LIN {X 0,Y 549.167,Z 589.017,A -85,B 0,C 180,E1 -11279.852,E2 -11279.852} C_VEL
LIN {X 0,Y 549.143,Z 589.013,A -85,B 0,C 180,E1 -11282.665,E2 -11282.665} C_VEL
LIN {X 0,Y 549.213,Z 589.004,A -85,B 0,C 180,E1 -11285.921,E2 -11285.921} C_VEL
LIN {X 0,Y 549.155,Z 589.006,A -85,B 0,C 180,E1 -11288.918,E2 -11288.918} C_VEL
LIN {X 0,Y 549.152,Z 589.01,A -85,B 0,C 180,E1 -11291.549,E2 -11291.549} C_VEL
LIN {X 0,Y 549.201,Z 589.004,A -85,B 0,C 180,E1 -11294.545,E2 -11294.545} C_VEL
LIN {X 0,Y 549.18,Z 589.01,A -85,B 0,C 180,E1 -11297.711,E2 -11297.711} C_VEL
LIN {X 0,Y 549.182,Z 589.007,A -85,B 0,C 180,E1 -11300.378,E2 -11300.378} C_VEL
LIN {X 0,Y 549.209,Z 589.006,A -85,B 0,C 180,E1 -11303.464,E2 -11303.464} C_VEL
LIN {X 0,Y 549.192,Z 589.005,A -85,B 0,C 180,E1 -11305.998,E2 -11305.998} C_VEL
LIN {X 0,Y 549.178,Z 589.011,A -85,B 0,C 180,E1 -11308.71,E2 -11308.71} C_VEL
LIN {X 0,Y 549.192,Z 589.009,A -85,B 0,C 180,E1 -11311.01,E2 -11311.01} C_VEL
LIN {X 0,Y 549.177,Z 589.009,A -85,B 0,C 180,E1 -11313.487,E2 -11313.487} C_VEL
LIN {X 0,Y 549.182,Z 589.008,A -85,B 0,C 180,E1 -11315.912,E2 -11315.912} C_VEL
LIN {X 0,Y 549.213,Z 589.011,A -85,B 0,C 180,E1 -11318.594,E2 -11318.594} C_VEL
LIN {X 0,Y 549.193,Z 589.011,A -85,B 0,C 180,E1 -11321.406,E2 -11321.406} C_VEL
LIN {X 0,Y 549.206,Z 589.008,A -85,B 0,C 180,E1 -11323.705,E2 -11323.705} C_VEL
LIN {X 0,Y 549.285,Z 588.998,A -85,B 0,C 180,E1 -11325.978,E2 -11325.978} C_VEL
LIN {X 0,Y 549.266,Z 589.108,A -85,B 0,C 180,E1 -11328.087,E2 -11328.087} C_VEL
LIN {X 0,Y 551,Z 598.292,A -85,B 0,C 180,E1 -11330.118,E2 -11330.118} C_VEL
LIN {X 0,Y 551.12,Z 603.64,A -85,B 0,C 180,E1 -11331.227,E2 -11331.227} C_VEL
LIN {X 0,Y 550.41,Z 616.517,A -85,B 0,C 180,E1 -11333.79,E2 -11333.79} C_VEL
LIN {X 0,Y 549.829,Z 624.477,A -85,B 0,C 180,E1 -11335.341,E2 -11335.341} C_VEL
LIN {X 0,Y 553.064,Z 642.479,A -85,B 0,C 180,E1 -11335.755,E2 -11335.755} C_VEL
LIN {X 0,Y 551.552,Z 730.311,A -85,B 0,C 180,E1 -11337.111,E2 -11337.111} C_VEL
LIN {X 0,Y 551.333,Z 739.943,A -85,B 0,C 180,E1 -11337.337,E2 -11337.337} C_VEL
LIN {X 0,Y 551.078,Z 750.352,A -85,B 0,C 180,E1 -11337.678,E2 -11337.678} C_VEL
LIN {X 0,Y 550.845,Z 759.981,A -85,B 0,C 180,E1 -11338.087,E2 -11338.087} C_VEL
LIN {X 0,Y 550.538,Z 770.195,A -85,B 0,C 180,E1 -11338.633,E2 -11338.633} C_VEL
LIN {X 0,Y 550.186,Z 779.879,A -85,B 0,C 180,E1 -11339.27,E2 -11339.27} C_VEL
LIN {X 0,Y 549.809,Z 788.022,A -85,B 0,C 180,E1 -11339.909,E2 -11339.909} C_VEL
LIN {X 0,Y 549.317,Z 796.766,A -85,B 0,C 180,E1 -11340.73,E2 -11340.73} C_VEL
LIN {X 0,Y 548.892,Z 803.411,A -85,B 0,C 180,E1 -11341.462,E2 -11341.462} C_VEL
LIN {X 0,Y 548.614,Z 810.348,A -85,B 0,C 180,E1 -11342.378,E2 -11342.378} C_VEL
LIN {X 0,Y 548.231,Z 816.184,A -85,B 0,C 180,E1 -11343.296,E2 -11343.296} C_VEL
LIN {X 0,Y 548.099,Z 822.583,A -85,B 0,C 180,E1 -11344.579,E2 -11344.579} C_VEL
LIN {X 0,Y 547.955,Z 827.199,A -85,B 0,C 180,E1 -11345.793,E2 -11345.793} C_VEL
LIN {X 0,Y 547.864,Z 829.635,A -85,B 0,C 180,E1 -11346.607,E2 -11346.607} C_VEL
LIN {X 0,Y 547.753,Z 831.287,A -85,B 0,C 180,E1 -11347.347,E2 -11347.347} C_VEL
LIN {X 0,Y 547.692,Z 833.366,A -85,B 0,C 180,E1 -11348.828,E2 -11348.828} C_VEL
LIN {X 0,Y 547.683,Z 833.621,A -85,B 0,C 180,E1 -11350.314,E2 -11350.314} C_VEL
LIN {X 0,Y 547.698,Z 833.236,A -85,B 0,C 180,E1 -11351.059,E2 -11351.059} C_VEL
LIN {X 0,Y 547.699,Z 830.896,A -85,B 0,C 180,E1 -11352.557,E2 -11352.557} C_VEL
LIN {X 0,Y 547.84,Z 828.07,A -85,B 0,C 180,E1 -11353.662,E2 -11353.662} C_VEL
LIN {X 0,Y 547.893,Z 825.548,A -85,B 0,C 180,E1 -11354.435,E2 -11354.435} C_VEL
LIN {X 0,Y 548.091,Z 819.726,A -85,B 0,C 180,E1 -11355.757,E2 -11355.757} C_VEL
LIN {X 0,Y 548.25,Z 814.051,A -85,B 0,C 180,E1 -11356.773,E2 -11356.773} C_VEL
LIN {X 0,Y 548.469,Z 808.116,A -85,B 0,C 180,E1 -11357.656,E2 -11357.656} C_VEL
LIN {X 0,Y 548.826,Z 800.373,A -85,B 0,C 180,E1 -11358.606,E2 -11358.606} C_VEL
LIN {X 0,Y 549.141,Z 791.937,A -85,B 0,C 180,E1 -11359.465,E2 -11359.465} C_VEL
LIN {X 0,Y 549.465,Z 782.896,A -85,B 0,C 180,E1 -11360.229,E2 -11360.229} C_VEL
LIN {X 0,Y 549.851,Z 773.343,A -85,B 0,C 180,E1 -11360.896,E2 -11360.896} C_VEL
LIN {X 0,Y 550.162,Z 765.257,A -85,B 0,C 180,E1 -11361.373,E2 -11361.373} C_VEL
LIN {X 0,Y 550.473,Z 753.781,A -85,B 0,C 180,E1 -11361.91,E2 -11361.91} C_VEL
LIN {X 0,Y 550.673,Z 742.561,A -85,B 0,C 180,E1 -11362.31,E2 -11362.31} C_VEL
LIN {X 0,Y 550.9,Z 732.608,A -85,B 0,C 180,E1 -11362.57,E2 -11362.57} C_VEL
LIN {X 0,Y 551.202,Z 713.558,A -85,B 0,C 180,E1 -11362.878,E2 -11362.878} C_VEL
LIN {X 0,Y 551.969,Z 640.723,A -85,B 0,C 180,E1 -11363.953,E2 -11363.953} C_VEL
LIN {X 0,Y 549.342,Z 623.321,A -85,B 0,C 180,E1 -11364.283,E2 -11364.283} C_VEL
LIN {X 0,Y 550.029,Z 607.305,A -85,B 0,C 180,E1 -11367.287,E2 -11367.287} C_VEL
LIN {X 0,Y 550.372,Z 596.511,A -85,B 0,C 180,E1 -11369.339,E2 -11369.339} C_VEL
LIN {X 0,Y 549.276,Z 588.999,A -85,B 0,C 180,E1 -11370.871,E2 -11370.871} C_VEL
LIN {X 0,Y 549.193,Z 589.009,A -85,B 0,C 180,E1 -11374.137,E2 -11374.137} C_VEL
LIN {X 0,Y 549.19,Z 589.003,A -85,B 0,C 180,E1 -11376.83,E2 -11376.83} C_VEL
LIN {X 0,Y 549.2,Z 589.009,A -85,B 0,C 180,E1 -11380.072,E2 -11380.072} C_VEL
LIN {X 0,Y 549.187,Z 589.005,A -85,B 0,C 180,E1 -11383.365,E2 -11383.365} C_VEL
LIN {X 0,Y 549.195,Z 589.006,A -85,B 0,C 180,E1 -11385.579,E2 -11385.579} C_VEL
LIN {X 0,Y 549.173,Z 589.005,A -85,B 0,C 180,E1 -11388.808,E2 -11388.808} C_VEL
LIN {X 0,Y 549.149,Z 589.009,A -85,B 0,C 180,E1 -11391.318,E2 -11391.318} C_VEL
LIN {X 0,Y 549.236,Z 589.005,A -85,B 0,C 180,E1 -11394.081,E2 -11394.081} C_VEL
LIN {X 0,Y 549.162,Z 589.007,A -85,B 0,C 180,E1 -11396.739,E2 -11396.739} C_VEL
LIN {X 0,Y 549.177,Z 589.005,A -85,B 0,C 180,E1 -11399.324,E2 -11399.324} C_VEL
LIN {X 0,Y 549.202,Z 589.009,A -85,B 0,C 180,E1 -11401.843,E2 -11401.843} C_VEL
LIN {X 0,Y 549.169,Z 589.005,A -85,B 0,C 180,E1 -11404.9,E2 -11404.9} C_VEL
LIN {X 0,Y 549.197,Z 589.005,A -85,B 0,C 180,E1 -11407.504,E2 -11407.504} C_VEL
LIN {X 0,Y 549.19,Z 589.01,A -85,B 0,C 180,E1 -11409.857,E2 -11409.857} C_VEL
LIN {X 0,Y 549.225,Z 588.998,A -85,B 0,C 180,E1 -11413.036,E2 -11413.036} C_VEL
LIN {X 0,Y 549.283,Z 589.001,A -85,B 0,C 180,E1 -11415.978,E2 -11415.978} C_VEL
LIN {X 0,Y 549.241,Z 588.998,A -85,B 0,C 180,E1 -11416.542,E2 -11416.542} C_VEL
LIN {X 0,Y 548.584,Z 589.079,A -85,B 0,C 180,E1 -11417.154,E2 -11417.154} C_VEL
LIN {X 0,Y 545.779,Z 589.434,A -85,B 0,C 180,E1 -11418.148,E2 -11418.148} C_VEL
LIN {X 0,Y 543.388,Z 589.731,A -85,B 0,C 180,E1 -11418.948,E2 -11418.948} C_VEL
LIN {X 0,Y 542.33,Z 589.861,A -85,B 0,C 180,E1 -11419.565,E2 -11419.565} C_VEL
LIN {X 0,Y 542.226,Z 589.873,A -85,B 0,C 180,E1 -11419.774,E2 -11419.774} C_VEL
LIN {X 0,Y 542.282,Z 589.865,A -85,B 0,C 180,E1 -11422.578,E2 -11422.578} C_VEL
LIN {X 0,Y 542.347,Z 589.855,A -85,B 0,C 180,E1 -11424.813,E2 -11424.813} C_VEL
LIN {X 0,Y 542.15,Z 589.88,A -85,B 0,C 180,E1 -11427.038,E2 -11427.038} C_VEL
LIN {X 0,Y 542.498,Z 589.846,A -85,B 0,C 180,E1 -11430,E2 -11430} C_VEL
LIN {X 0,Y 542.313,Z 589.865,A -85,B 0,C 180,E1 -11433.703,E2 -11433.703} C_VEL
LIN {X 0,Y 542.34,Z 589.865,A -85,B 0,C 180,E1 -11436.033,E2 -11436.033} C_VEL
LIN {X 0,Y 542.226,Z 589.87,A -85,B 0,C 180,E1 -11438.918,E2 -11438.918} C_VEL
LIN {X 0,Y 542.235,Z 589.869,A -85,B 0,C 180,E1 -11441.173,E2 -11441.173} C_VEL
LIN {X 0,Y 542.236,Z 589.873,A -85,B 0,C 180,E1 -11444.346,E2 -11444.346} C_VEL
LIN {X 0,Y 542.17,Z 589.878,A -85,B 0,C 180,E1 -11447.286,E2 -11447.286} C_VEL
LIN {X 0,Y 542.161,Z 589.881,A -85,B 0,C 180,E1 -11450.415,E2 -11450.415} C_VEL
LIN {X 0,Y 542.138,Z 589.881,A -85,B 0,C 180,E1 -11452.805,E2 -11452.805} C_VEL
LIN {X 0,Y 542.134,Z 589.882,A -85,B 0,C 180,E1 -11455.258,E2 -11455.258} C_VEL
LIN {X 0,Y 542.151,Z 589.885,A -85,B 0,C 180,E1 -11457.717,E2 -11457.717} C_VEL
LIN {X 0,Y 542.149,Z 589.885,A -85,B 0,C 180,E1 -11460.256,E2 -11460.256} C_VEL
LIN {X 0,Y 542.129,Z 589.882,A -85,B 0,C 180,E1 -11462.88,E2 -11462.88} C_VEL
LIN {X 0,Y 542.188,Z 589.878,A -85,B 0,C 180,E1 -11465.545,E2 -11465.545} C_VEL
LIN {X 0,Y 542.123,Z 589.887,A -85,B 0,C 180,E1 -11468.329,E2 -11468.329} C_VEL
LIN {X 0,Y 542.125,Z 589.883,A -85,B 0,C 180,E1 -11471.219,E2 -11471.219} C_VEL
LIN {X 0,Y 542.15,Z 589.885,A -85,B 0,C 180,E1 -11474.24,E2 -11474.24} C_VEL
LIN {X 0,Y 542.127,Z 589.883,A -85,B 0,C 180,E1 -11476.783,E2 -11476.783} C_VEL
LIN {X 0,Y 542.153,Z 589.885,A -85,B 0,C 180,E1 -11479.761,E2 -11479.761} C_VEL
LIN {X 0,Y 542.165,Z 589.879,A -85,B 0,C 180,E1 -11482.612,E2 -11482.612} C_VEL
LIN {X 0,Y 542.155,Z 589.881,A -85,B 0,C 180,E1 -11485.357,E2 -11485.357} C_VEL
LIN {X 0,Y 542.125,Z 589.885,A -85,B 0,C 180,E1 -11488.511,E2 -11488.511} C_VEL
LIN {X 0,Y 542.142,Z 589.883,A -85,B 0,C 180,E1 -11491.468,E2 -11491.468} C_VEL
LIN {X 0,Y 542.111,Z 589.894,A -85,B 0,C 180,E1 -11493.941,E2 -11493.941} C_VEL
LIN {X 0,Y 542.138,Z 589.883,A -85,B 0,C 180,E1 -11496.538,E2 -11496.538} C_VEL
LIN {X 0,Y 542.165,Z 589.878,A -85,B 0,C 180,E1 -11498.793,E2 -11498.793} C_VEL
LIN {X 0,Y 542.15,Z 589.88,A -85,B 0,C 180,E1 -11501.156,E2 -11501.156} C_VEL
LIN {X 0,Y 542.164,Z 589.881,A -85,B 0,C 180,E1 -11503.488,E2 -11503.488} C_VEL
LIN {X 0,Y 542.242,Z 589.875,A -85,B 0,C 180,E1 -11505.793,E2 -11505.793} C_VEL
LIN {X 0,Y 542.279,Z 589.864,A -85,B 0,C 180,E1 -11509.012,E2 -11509.012} C_VEL
LIN {X 0,Y 542.263,Z 589.873,A -85,B 0,C 180,E1 -11511.832,E2 -11511.832} C_VEL
LIN {X 0,Y 542.352,Z 589.862,A -85,B 0,C 180,E1 -11514.07,E2 -11514.07} C_VEL
LIN {X 0,Y 542.308,Z 589.864,A -85,B 0,C 180,E1 -11516.298,E2 -11516.298} C_VEL
LIN {X 0,Y 542.502,Z 589.845,A -85,B 0,C 180,E1 -11520,E2 -11520} C_VEL
LIN {X 0,Y 542.306,Z 589.866,A -85,B 0,C 180,E1 -11523.703,E2 -11523.703} C_VEL
LIN {X 0,Y 542.364,Z 589.861,A -85,B 0,C 180,E1 -11526.052,E2 -11526.052} C_VEL
LIN {X 0,Y 542.233,Z 589.869,A -85,B 0,C 180,E1 -11528.918,E2 -11528.918} C_VEL
LIN {X 0,Y 542.238,Z 589.869,A -85,B 0,C 180,E1 -11531.173,E2 -11531.173} C_VEL
LIN {X 0,Y 542.227,Z 589.874,A -85,B 0,C 180,E1 -11534.34,E2 -11534.34} C_VEL
LIN {X 0,Y 542.136,Z 589.883,A -85,B 0,C 180,E1 -11537.287,E2 -11537.287} C_VEL
LIN {X 0,Y 542.139,Z 589.885,A -85,B 0,C 180,E1 -11539.629,E2 -11539.629} C_VEL
LIN {X 0,Y 542.124,Z 589.892,A -85,B 0,C 180,E1 -11542.005,E2 -11542.005} C_VEL
LIN {X 0,Y 542.137,Z 589.884,A -85,B 0,C 180,E1 -11544.421,E2 -11544.421} C_VEL
LIN {X 0,Y 542.154,Z 589.885,A -85,B 0,C 180,E1 -11547.717,E2 -11547.717} C_VEL
LIN {X 0,Y 542.121,Z 589.888,A -85,B 0,C 180,E1 -11550.258,E2 -11550.258} C_VEL
LIN {X 0,Y 542.112,Z 589.885,A -85,B 0,C 180,E1 -11552.877,E2 -11552.877} C_VEL
LIN {X 0,Y 542.121,Z 589.887,A -85,B 0,C 180,E1 -11555.55,E2 -11555.55} C_VEL
LIN {X 0,Y 542.088,Z 589.891,A -85,B 0,C 180,E1 -11558.332,E2 -11558.332} C_VEL
LIN {X 0,Y 542.13,Z 589.885,A -85,B 0,C 180,E1 -11561.464,E2 -11561.464} C_VEL
LIN {X 0,Y 542.149,Z 589.88,A -85,B 0,C 180,E1 -11564.717,E2 -11564.717} C_VEL
LIN {X 0,Y 542.103,Z 589.888,A -85,B 0,C 180,E1 -11567.433,E2 -11567.433} C_VEL
LIN {X 0,Y 542.116,Z 589.89,A -85,B 0,C 180,E1 -11569.757,E2 -11569.757} C_VEL
LIN {X 0,Y 542.1,Z 589.887,A -85,B 0,C 180,E1 -11572.607,E2 -11572.607} C_VEL
LIN {X 0,Y 542.12,Z 589.885,A -85,B 0,C 180,E1 -11575.354,E2 -11575.354} C_VEL
LIN {X 0,Y 542.109,Z 589.894,A -85,B 0,C 180,E1 -11578.012,E2 -11578.012} C_VEL
LIN {X 0,Y 542.139,Z 589.882,A -85,B 0,C 180,E1 -11580.596,E2 -11580.596} C_VEL
LIN {X 0,Y 542.116,Z 589.884,A -85,B 0,C 180,E1 -11583.114,E2 -11583.114} C_VEL
LIN {X 0,Y 542.153,Z 589.943,A -85,B 0,C 180,E1 -11585.935,E2 -11585.935} C_VEL
LIN {X 0,Y 544.262,Z 601.967,A -85,B 0,C 180,E1 -11588.086,E2 -11588.086} C_VEL
LIN {X 0,Y 543.789,Z 613.914,A -85,B 0,C 180,E1 -11590.102,E2 -11590.102} C_VEL
LIN {X 0,Y 542.762,Z 634.369,A -85,B 0,C 180,E1 -11593.506,E2 -11593.506} C_VEL
LIN {X 0,Y 542.247,Z 647.24,A -85,B 0,C 180,E1 -11595.592,E2 -11595.592} C_VEL
LIN {X 0,Y 544.925,Z 670.18,A -85,B 0,C 180,E1 -11596.006,E2 -11596.006} C_VEL
LIN {X 0,Y 543.974,Z 754.194,A -85,B 0,C 180,E1 -11597.285,E2 -11597.285} C_VEL
LIN {X 0,Y 543.75,Z 763.983,A -85,B 0,C 180,E1 -11597.516,E2 -11597.516} C_VEL
LIN {X 0,Y 543.475,Z 773.356,A -85,B 0,C 180,E1 -11597.817,E2 -11597.817} C_VEL
LIN {X 0,Y 543.155,Z 784.221,A -85,B 0,C 180,E1 -11598.277,E2 -11598.277} C_VEL
LIN {X 0,Y 542.941,Z 792.736,A -85,B 0,C 180,E1 -11598.722,E2 -11598.722} C_VEL
LIN {X 0,Y 542.524,Z 803.182,A -85,B 0,C 180,E1 -11599.398,E2 -11599.398} C_VEL
LIN {X 0,Y 542.148,Z 812.599,A -85,B 0,C 180,E1 -11600.143,E2 -11600.143} C_VEL
LIN {X 0,Y 541.76,Z 820.502,A -85,B 0,C 180,E1 -11600.887,E2 -11600.887} C_VEL
LIN {X 0,Y 541.379,Z 828.715,A -85,B 0,C 180,E1 -11601.818,E2 -11601.818} C_VEL
LIN {X 0,Y 541.142,Z 835.553,A -85,B 0,C 180,E1 -11602.75,E2 -11602.75} C_VEL
LIN {X 0,Y 540.958,Z 841.257,A -85,B 0,C 180,E1 -11603.681,E2 -11603.681} C_VEL
LIN {X 0,Y 540.832,Z 846.778,A -85,B 0,C 180,E1 -11604.799,E2 -11604.799} C_VEL
LIN {X 0,Y 540.736,Z 849.867,A -85,B 0,C 180,E1 -11605.543,E2 -11605.543} C_VEL
LIN {X 0,Y 540.68,Z 853.432,A -85,B 0,C 180,E1 -11606.658,E2 -11606.658} C_VEL
LIN {X 0,Y 540.682,Z 855.954,A -85,B 0,C 180,E1 -11607.773,E2 -11607.773} C_VEL
LIN {X 0,Y 540.646,Z 857.752,A -85,B 0,C 180,E1 -11609.258,E2 -11609.258} C_VEL
LIN {X 0,Y 540.635,Z 858.065,A -85,B 0,C 180,E1 -11610,E2 -11610} C_VEL
LIN {X 0,Y 540.647,Z 857.414,A -85,B 0,C 180,E1 -11611.485,E2 -11611.485} C_VEL
LIN {X 0,Y 540.682,Z 856.4,A -85,B 0,C 180,E1 -11612.227,E2 -11612.227} C_VEL
LIN {X 0,Y 540.712,Z 853.243,A -85,B 0,C 180,E1 -11613.714,E2 -11613.714} C_VEL
LIN {X 0,Y 540.783,Z 849.623,A -85,B 0,C 180,E1 -11614.83,E2 -11614.83} C_VEL
LIN {X 0,Y 540.937,Z 844.88,A -85,B 0,C 180,E1 -11615.946,E2 -11615.946} C_VEL
LIN {X 0,Y 541.151,Z 838.85,A -85,B 0,C 180,E1 -11617.063,E2 -11617.063} C_VEL
LIN {X 0,Y 541.488,Z 831.311,A -85,B 0,C 180,E1 -11618.181,E2 -11618.181} C_VEL
LIN {X 0,Y 541.88,Z 823.679,A -85,B 0,C 180,E1 -11619.111,E2 -11619.111} C_VEL
LIN {X 0,Y 542.348,Z 815.452,A -85,B 0,C 180,E1 -11619.947,E2 -11619.947} C_VEL
LIN {X 0,Y 542.781,Z 806.721,A -85,B 0,C 180,E1 -11620.691,E2 -11620.691} C_VEL
LIN {X 0,Y 543.202,Z 797.041,A -85,B 0,C 180,E1 -11621.375,E2 -11621.375} C_VEL
LIN {X 0,Y 543.603,Z 788.118,A -85,B 0,C 180,E1 -11621.898,E2 -11621.898} C_VEL
LIN {X 0,Y 544.02,Z 777.27,A -85,B 0,C 180,E1 -11622.407,E2 -11622.407} C_VEL
LIN {X 0,Y 544.358,Z 767.174,A -85,B 0,C 180,E1 -11622.777,E2 -11622.777} C_VEL
LIN {X 0,Y 544.713,Z 755.878,A -85,B 0,C 180,E1 -11623.076,E2 -11623.076} C_VEL
LIN {X 0,Y 545.07,Z 733.637,A -85,B 0,C 180,E1 -11623.445,E2 -11623.445} C_VEL
LIN {X 0,Y 545.976,Z 669.088,A -85,B 0,C 180,E1 -11624.461,E2 -11624.461} C_VEL
LIN {X 0,Y 543.573,Z 651.51,A -85,B 0,C 180,E1 -11624.84,E2 -11624.84} C_VEL
LIN {X 0,Y 542.613,Z 645.876,A -85,B 0,C 180,E1 -11624.986,E2 -11624.986} C_VEL
LIN {X 0,Y 543.607,Z 626.95,A -85,B 0,C 180,E1 -11628.208,E2 -11628.208} C_VEL
LIN {X 0,Y 544.885,Z 608.18,A -85,B 0,C 180,E1 -11631.492,E2 -11631.492} C_VEL
LIN {X 0,Y 544.87,Z 604.061,A -85,B 0,C 180,E1 -11632.244,E2 -11632.244} C_VEL
LIN {X 0,Y 542.428,Z 591.113,A -85,B 0,C 180,E1 -11634.814,E2 -11634.814} C_VEL
LIN {X 0,Y 542.136,Z 589.89,A -85,B 0,C 180,E1 -11635.104,E2 -11635.104} C_VEL
LIN {X 0,Y 542.131,Z 589.895,A -85,B 0,C 180,E1 -11637.719,E2 -11637.719} C_VEL
LIN {X 0,Y 542.121,Z 589.89,A -85,B 0,C 180,E1 -11640.258,E2 -11640.258} C_VEL
LIN {X 0,Y 542.113,Z 589.89,A -85,B 0,C 180,E1 -11642.877,E2 -11642.877} C_VEL
LIN {X 0,Y 542.164,Z 589.885,A -85,B 0,C 180,E1 -11645.547,E2 -11645.547} C_VEL
LIN {X 0,Y 542.102,Z 589.883,A -85,B 0,C 180,E1 -11648.331,E2 -11648.331} C_VEL
LIN {X 0,Y 542.133,Z 589.884,A -85,B 0,C 180,E1 -11651.464,E2 -11651.464} C_VEL
LIN {X 0,Y 542.154,Z 589.881,A -85,B 0,C 180,E1 -11654.24,E2 -11654.24} C_VEL
LIN {X 0,Y 542.156,Z 589.885,A -85,B 0,C 180,E1 -11656.785,E2 -11656.785} C_VEL
LIN {X 0,Y 542.157,Z 589.883,A -85,B 0,C 180,E1 -11659.761,E2 -11659.761} C_VEL
LIN {X 0,Y 542.168,Z 589.886,A -85,B 0,C 180,E1 -11663.226,E2 -11663.226} C_VEL
LIN {X 0,Y 542.147,Z 589.883,A -85,B 0,C 180,E1 -11665.779,E2 -11665.779} C_VEL
LIN {X 0,Y 542.128,Z 589.892,A -85,B 0,C 180,E1 -11668.881,E2 -11668.881} C_VEL
LIN {X 0,Y 542.146,Z 589.884,A -85,B 0,C 180,E1 -11671.468,E2 -11671.468} C_VEL
LIN {X 0,Y 542.112,Z 589.889,A -85,B 0,C 180,E1 -11673.941,E2 -11673.941} C_VEL
LIN {X 0,Y 542.143,Z 589.891,A -85,B 0,C 180,E1 -11676.537,E2 -11676.537} C_VEL
LIN {X 0,Y 542.164,Z 589.885,A -85,B 0,C 180,E1 -11679.584,E2 -11679.584} C_VEL
LIN {X 0,Y 542.155,Z 589.889,A -85,B 0,C 180,E1 -11681.936,E2 -11681.936} C_VEL
LIN {X 0,Y 542.206,Z 589.88,A -85,B 0,C 180,E1 -11685.027,E2 -11685.027} C_VEL
LIN {X 0,Y 542.244,Z 589.98,A -85,B 0,C 180,E1 -11687.835,E2 -11687.835} C_VEL
LIN {X 0,Y 544.06,Z 599.517,A -85,B 0,C 180,E1 -11689.991,E2 -11689.991} C_VEL
LIN {X 0,Y 544.203,Z 604.855,A -85,B 0,C 180,E1 -11691.115,E2 -11691.115} C_VEL
LIN {X 0,Y 543.453,Z 617.675,A -85,B 0,C 180,E1 -11693.71,E2 -11693.71} C_VEL
LIN {X 0,Y 542.906,Z 624.687,A -85,B 0,C 180,E1 -11695.097,E2 -11695.097} C_VEL
LIN {X 0,Y 546.289,Z 642.987,A -85,B 0,C 180,E1 -11695.53,E2 -11695.53} C_VEL
LIN {X 0,Y 545.008,Z 710.544,A -85,B 0,C 180,E1 -11696.592,E2 -11696.592} C_VEL
LIN {X 0,Y 544.667,Z 732.534,A -85,B 0,C 180,E1 -11696.959,E2 -11696.959} C_VEL
LIN {X 0,Y 544.359,Z 745.377,A -85,B 0,C 180,E1 -11697.303,E2 -11697.303} C_VEL
LIN {X 0,Y 543.974,Z 759.583,A -85,B 0,C 180,E1 -11697.878,E2 -11697.878} C_VEL
LIN {X 0,Y 543.646,Z 769.909,A -85,B 0,C 180,E1 -11698.431,E2 -11698.431} C_VEL
LIN {X 0,Y 543.309,Z 779.666,A -85,B 0,C 180,E1 -11699.076,E2 -11699.076} C_VEL
LIN {X 0,Y 542.822,Z 788.904,A -85,B 0,C 180,E1 -11699.815,E2 -11699.815} C_VEL
LIN {X 0,Y 542.376,Z 796.687,A -85,B 0,C 180,E1 -11700.555,E2 -11700.555} C_VEL
LIN {X 0,Y 541.835,Z 804.804,A -85,B 0,C 180,E1 -11701.481,E2 -11701.481} C_VEL
LIN {X 0,Y 541.545,Z 811.542,A -85,B 0,C 180,E1 -11702.409,E2 -11702.409} C_VEL
LIN {X 0,Y 541.159,Z 817.201,A -85,B 0,C 180,E1 -11703.339,E2 -11703.339} C_VEL
LIN {X 0,Y 541.067,Z 822.652,A -85,B 0,C 180,E1 -11704.455,E2 -11704.455} C_VEL
LIN {X 0,Y 540.901,Z 826.94,A -85,B 0,C 180,E1 -11705.573,E2 -11705.573} C_VEL
LIN {X 0,Y 540.76,Z 830.153,A -85,B 0,C 180,E1 -11706.694,E2 -11706.694} C_VEL
LIN {X 0,Y 540.644,Z 831.8,A -85,B 0,C 180,E1 -11707.444,E2 -11707.444} C_VEL
LIN {X 0,Y 540.593,Z 833.6,A -85,B 0,C 180,E1 -11708.945,E2 -11708.945} C_VEL
LIN {X 0,Y 540.618,Z 833.9,A -85,B 0,C 180,E1 -11710.039,E2 -11710.039} C_VEL
LIN {X 0,Y 540.601,Z 833.202,A -85,B 0,C 180,E1 -11711.207,E2 -11711.207} C_VEL
LIN {X 0,Y 540.556,Z 832.172,A -85,B 0,C 180,E1 -11711.965,E2 -11711.965} C_VEL
LIN {X 0,Y 540.733,Z 828.837,A -85,B 0,C 180,E1 -11713.483,E2 -11713.483} C_VEL
LIN {X 0,Y 540.825,Z 825.024,A -85,B 0,C 180,E1 -11714.628,E2 -11714.628} C_VEL
LIN {X 0,Y 541.005,Z 819.977,A -85,B 0,C 180,E1 -11715.776,E2 -11715.776} C_VEL
LIN {X 0,Y 541.159,Z 814.982,A -85,B 0,C 180,E1 -11716.701,E2 -11716.701} C_VEL
LIN {X 0,Y 541.399,Z 808.392,A -85,B 0,C 180,E1 -11717.7,E2 -11717.7} C_VEL
LIN {X 0,Y 541.758,Z 800.663,A -85,B 0,C 180,E1 -11718.662,E2 -11718.662} C_VEL
LIN {X 0,Y 542.075,Z 793.055,A -85,B 0,C 180,E1 -11719.459,E2 -11719.459} C_VEL
LIN {X 0,Y 542.412,Z 783.227,A -85,B 0,C 180,E1 -11720.307,E2 -11720.307} C_VEL
LIN {X 0,Y 542.831,Z 773.716,A -85,B 0,C 180,E1 -11720.982,E2 -11720.982} C_VEL
LIN {X 0,Y 543.155,Z 764.302,A -85,B 0,C 180,E1 -11721.534,E2 -11721.534} C_VEL
LIN {X 0,Y 543.475,Z 754.567,A -85,B 0,C 180,E1 -11721.997,E2 -11721.997} C_VEL
LIN {X 0,Y 543.669,Z 743.239,A -85,B 0,C 180,E1 -11722.412,E2 -11722.412} C_VEL
LIN {X 0,Y 543.91,Z 732.23,A -85,B 0,C 180,E1 -11722.701,E2 -11722.701} C_VEL
LIN {X 0,Y 544.239,Z 713.189,A -85,B 0,C 180,E1 -11723.012,E2 -11723.012} C_VEL
LIN {X 0,Y 545.027,Z 641.328,A -85,B 0,C 180,E1 -11724.09,E2 -11724.09} C_VEL
LIN {X 0,Y 542.333,Z 623.472,A -85,B 0,C 180,E1 -11724.437,E2 -11724.437} C_VEL
LIN {X 0,Y 543.008,Z 608.118,A -85,B 0,C 180,E1 -11727.349,E2 -11727.349} C_VEL
LIN {X 0,Y 543.387,Z 597.81,A -85,B 0,C 180,E1 -11729.329,E2 -11729.329} C_VEL
LIN {X 0,Y 542.233,Z 589.876,A -85,B 0,C 180,E1 -11730.949,E2 -11730.949} C_VEL
LIN {X 0,Y 542.145,Z 589.886,A -85,B 0,C 180,E1 -11734.221,E2 -11734.221} C_VEL
LIN {X 0,Y 542.165,Z 589.878,A -85,B 0,C 180,E1 -11736.774,E2 -11736.774} C_VEL
LIN {X 0,Y 542.154,Z 589.884,A -85,B 0,C 180,E1 -11740.239,E2 -11740.239} C_VEL
LIN {X 0,Y 542.129,Z 589.883,A -85,B 0,C 180,E1 -11743.217,E2 -11743.217} C_VEL
LIN {X 0,Y 542.152,Z 589.885,A -85,B 0,C 180,E1 -11745.76,E2 -11745.76} C_VEL
LIN {X 0,Y 542.127,Z 589.883,A -85,B 0,C 180,E1 -11748.781,E2 -11748.781} C_VEL
LIN {X 0,Y 542.099,Z 589.891,A -85,B 0,C 180,E1 -11751.669,E2 -11751.669} C_VEL
LIN {X 0,Y 542.19,Z 589.877,A -85,B 0,C 180,E1 -11754.476,E2 -11754.476} C_VEL
LIN {X 0,Y 542.118,Z 589.884,A -85,B 0,C 180,E1 -11757.135,E2 -11757.135} C_VEL
LIN {X 0,Y 542.15,Z 589.889,A -85,B 0,C 180,E1 -11759.953,E2 -11759.953} C_VEL
LIN {X 0,Y 542.156,Z 589.879,A -85,B 0,C 180,E1 -11763.055,E2 -11763.055} C_VEL
LIN {X 0,Y 542.138,Z 589.885,A -85,B 0,C 180,E1 -11765.579,E2 -11765.579} C_VEL
LIN {X 0,Y 542.169,Z 589.88,A -85,B 0,C 180,E1 -11768.463,E2 -11768.463} C_VEL
LIN {X 0,Y 542.152,Z 589.88,A -85,B 0,C 180,E1 -11771.156,E2 -11771.156} C_VEL
LIN {X 0,Y 542.186,Z 589.878,A -85,B 0,C 180,E1 -11773.488,E2 -11773.488} C_VEL
LIN {X 0,Y 542.241,Z 589.875,A -85,B 0,C 180,E1 -11775.792,E2 -11775.792} C_VEL
LIN {X 0,Y 542.275,Z 589.864,A -85,B 0,C 180,E1 -11779.011,E2 -11779.011} C_VEL
LIN {X 0,Y 542.226,Z 589.873,A -85,B 0,C 180,E1 -11779.774,E2 -11779.774} C_VEL
LIN {X 0,Y 541.518,Z 589.962,A -85,B 0,C 180,E1 -11780.394,E2 -11780.394} C_VEL
LIN {X 0,Y 538.673,Z 590.315,A -85,B 0,C 180,E1 -11781.401,E2 -11781.401} C_VEL
LIN {X 0,Y 536.311,Z 590.613,A -85,B 0,C 180,E1 -11782.211,E2 -11782.211} C_VEL
LIN {X 0,Y 535.317,Z 590.731,A -85,B 0,C 180,E1 -11782.837,E2 -11782.837} C_VEL
LIN {X 0,Y 535.245,Z 590.74,A -85,B 0,C 180,E1 -11783.049,E2 -11783.049} C_VEL
LIN {X 0,Y 535.315,Z 590.734,A -85,B 0,C 180,E1 -11785.497,E2 -11785.497} C_VEL
LIN {X 0,Y 535.397,Z 590.722,A -85,B 0,C 180,E1 -11789.25,E2 -11789.25} C_VEL
LIN {X 0,Y 535.259,Z 590.741,A -85,B 0,C 180,E1 -11791.5,E2 -11791.5} C_VEL
LIN {X 0,Y 535.315,Z 590.733,A -85,B 0,C 180,E1 -11794.503,E2 -11794.503} C_VEL
LIN {X 0,Y 535.255,Z 590.739,A -85,B 0,C 180,E1 -11796.764,E2 -11796.764} C_VEL
LIN {X 0,Y 535.155,Z 590.758,A -85,B 0,C 180,E1 -11799.797,E2 -11799.797} C_VEL
LIN {X 0,Y 535.149,Z 590.759,A -85,B 0,C 180,E1 -11802.088,E2 -11802.088} C_VEL
LIN {X 0,Y 535.204,Z 590.748,A -85,B 0,C 180,E1 -11804.428,E2 -11804.428} C_VEL
LIN {X 0,Y 535.11,Z 590.76,A -85,B 0,C 180,E1 -11807.521,E2 -11807.521} C_VEL
LIN {X 0,Y 535.132,Z 590.755,A -85,B 0,C 180,E1 -11810.696,E2 -11810.696} C_VEL
LIN {X 0,Y 535.091,Z 590.763,A -85,B 0,C 180,E1 -11813.609,E2 -11813.609} C_VEL
LIN {X 0,Y 535.079,Z 590.763,A -85,B 0,C 180,E1 -11816.428,E2 -11816.428} C_VEL
LIN {X 0,Y 535.098,Z 590.758,A -85,B 0,C 180,E1 -11818.969,E2 -11818.969} C_VEL
LIN {X 0,Y 535.084,Z 590.765,A -85,B 0,C 180,E1 -11821.694,E2 -11821.694} C_VEL
LIN {X 0,Y 535.106,Z 590.76,A -85,B 0,C 180,E1 -11824.447,E2 -11824.447} C_VEL
LIN {X 0,Y 535.137,Z 590.753,A -85,B 0,C 180,E1 -11827.02,E2 -11827.02} C_VEL
LIN {X 0,Y 535.097,Z 590.767,A -85,B 0,C 180,E1 -11829.897,E2 -11829.897} C_VEL
LIN {X 0,Y 535.086,Z 590.76,A -85,B 0,C 180,E1 -11832.898,E2 -11832.898} C_VEL
LIN {X 0,Y 535.095,Z 590.759,A -85,B 0,C 180,E1 -11835.02,E2 -11835.02} C_VEL
LIN {X 0,Y 535.086,Z 590.76,A -85,B 0,C 180,E1 -11837.143,E2 -11837.143} C_VEL
LIN {X 0,Y 535.098,Z 590.765,A -85,B 0,C 180,E1 -11840.103,E2 -11840.103} C_VEL
LIN {X 0,Y 535.138,Z 590.753,A -85,B 0,C 180,E1 -11842.98,E2 -11842.98} C_VEL
LIN {X 0,Y 535.109,Z 590.763,A -85,B 0,C 180,E1 -11845.747,E2 -11845.747} C_VEL
LIN {X 0,Y 535.082,Z 590.763,A -85,B 0,C 180,E1 -11848.425,E2 -11848.425} C_VEL
LIN {X 0,Y 535.097,Z 590.759,A -85,B 0,C 180,E1 -11851.286,E2 -11851.286} C_VEL
LIN {X 0,Y 535.091,Z 590.763,A -85,B 0,C 180,E1 -11853.573,E2 -11853.573} C_VEL
LIN {X 0,Y 535.094,Z 590.762,A -85,B 0,C 180,E1 -11856.392,E2 -11856.392} C_VEL
LIN {X 0,Y 535.132,Z 590.755,A -85,B 0,C 180,E1 -11859.304,E2 -11859.304} C_VEL
LIN {X 0,Y 535.091,Z 590.764,A -85,B 0,C 180,E1 -11861.69,E2 -11861.69} C_VEL
LIN {X 0,Y 535.13,Z 590.762,A -85,B 0,C 180,E1 -11864.046,E2 -11864.046} C_VEL
LIN {X 0,Y 535.17,Z 590.753,A -85,B 0,C 180,E1 -11866.374,E2 -11866.374} C_VEL
LIN {X 0,Y 535.229,Z 590.744,A -85,B 0,C 180,E1 -11869.443,E2 -11869.443} C_VEL
LIN {X 0,Y 535.254,Z 590.741,A -85,B 0,C 180,E1 -11872.481,E2 -11872.481} C_VEL
LIN {X 0,Y 535.286,Z 590.735,A -85,B 0,C 180,E1 -11874.745,E2 -11874.745} C_VEL
LIN {X 0,Y 535.29,Z 590.739,A -85,B 0,C 180,E1 -11876.249,E2 -11876.249} C_VEL
LIN {X 0,Y 535.456,Z 590.723,A -85,B 0,C 180,E1 -11880,E2 -11880} C_VEL
LIN {X 0,Y 535.288,Z 590.74,A -85,B 0,C 180,E1 -11883.752,E2 -11883.752} C_VEL
LIN {X 0,Y 535.26,Z 590.738,A -85,B 0,C 180,E1 -11886.764,E2 -11886.764} C_VEL
LIN {X 0,Y 535.163,Z 590.757,A -85,B 0,C 180,E1 -11889.797,E2 -11889.797} C_VEL
LIN {X 0,Y 535.143,Z 590.76,A -85,B 0,C 180,E1 -11892.089,E2 -11892.089} C_VEL
LIN {X 0,Y 535.181,Z 590.751,A -85,B 0,C 180,E1 -11894.417,E2 -11894.417} C_VEL
LIN {X 0,Y 535.09,Z 590.762,A -85,B 0,C 180,E1 -11897.522,E2 -11897.522} C_VEL
LIN {X 0,Y 535.083,Z 590.768,A -85,B 0,C 180,E1 -11899.898,E2 -11899.898} C_VEL
LIN {X 0,Y 535.088,Z 590.763,A -85,B 0,C 180,E1 -11902.31,E2 -11902.31} C_VEL
LIN {X 0,Y 535.074,Z 590.762,A -85,B 0,C 180,E1 -11904.765,E2 -11904.765} C_VEL
LIN {X 0,Y 535.102,Z 590.759,A -85,B 0,C 180,E1 -11907.268,E2 -11907.268} C_VEL
LIN {X 0,Y 535.076,Z 590.766,A -85,B 0,C 180,E1 -11910.234,E2 -11910.234} C_VEL
LIN {X 0,Y 535.051,Z 590.765,A -85,B 0,C 180,E1 -11913.355,E2 -11913.355} C_VEL
LIN {X 0,Y 535.08,Z 590.768,A -85,B 0,C 180,E1 -11916.091,E2 -11916.091} C_VEL
LIN {X 0,Y 535.031,Z 590.767,A -85,B 0,C 180,E1 -11918.932,E2 -11918.932} C_VEL
LIN {X 0,Y 535.071,Z 590.77,A -85,B 0,C 180,E1 -11921.884,E2 -11921.884} C_VEL
LIN {X 0,Y 535.098,Z 590.758,A -85,B 0,C 180,E1 -11925.02,E2 -11925.02} C_VEL
LIN {X 0,Y 535.076,Z 590.766,A -85,B 0,C 180,E1 -11928.259,E2 -11928.259} C_VEL
LIN {X 0,Y 535.029,Z 590.767,A -85,B 0,C 180,E1 -11931.068,E2 -11931.068} C_VEL
LIN {X 0,Y 535.076,Z 590.77,A -85,B 0,C 180,E1 -11933.909,E2 -11933.909} C_VEL
LIN {X 0,Y 535.063,Z 590.763,A -85,B 0,C 180,E1 -11936.91,E2 -11936.91} C_VEL
LIN {X 0,Y 535.075,Z 590.767,A -85,B 0,C 180,E1 -11939.766,E2 -11939.766} C_VEL
LIN {X 0,Y 535.084,Z 590.76,A -85,B 0,C 180,E1 -11942.732,E2 -11942.732} C_VEL
LIN {X 0,Y 535.117,Z 590.902,A -85,B 0,C 180,E1 -11945.829,E2 -11945.829} C_VEL
LIN {X 0,Y 537.232,Z 602.351,A -85,B 0,C 180,E1 -11947.91,E2 -11947.91} C_VEL
LIN {X 0,Y 536.999,Z 610.905,A -85,B 0,C 180,E1 -11949.379,E2 -11949.379} C_VEL
LIN {X 0,Y 536.021,Z 628.236,A -85,B 0,C 180,E1 -11952.313,E2 -11952.313} C_VEL
LIN {X 0,Y 535.19,Z 646.849,A -85,B 0,C 180,E1 -11955.43,E2 -11955.43} C_VEL
LIN {X 0,Y 537.976,Z 670.747,A -85,B 0,C 180,E1 -11955.87,E2 -11955.87} C_VEL
LIN {X 0,Y 536.945,Z 753.056,A -85,B 0,C 180,E1 -11957.14,E2 -11957.14} C_VEL
LIN {X 0,Y 536.771,Z 763.169,A -85,B 0,C 180,E1 -11957.375,E2 -11957.375} C_VEL
LIN {X 0,Y 536.469,Z 773.301,A -85,B 0,C 180,E1 -11957.703,E2 -11957.703} C_VEL
LIN {X 0,Y 536.158,Z 783.671,A -85,B 0,C 180,E1 -11958.145,E2 -11958.145} C_VEL
LIN {X 0,Y 535.861,Z 793.802,A -85,B 0,C 180,E1 -11958.693,E2 -11958.693} C_VEL
LIN {X 0,Y 535.446,Z 803.696,A -85,B 0,C 180,E1 -11959.352,E2 -11959.352} C_VEL
LIN {X 0,Y 535.088,Z 811.971,A -85,B 0,C 180,E1 -11960.012,E2 -11960.012} C_VEL
LIN {X 0,Y 534.701,Z 819.955,A -85,B 0,C 180,E1 -11960.766,E2 -11960.766} C_VEL
LIN {X 0,Y 534.316,Z 828.24,A -85,B 0,C 180,E1 -11961.709,E2 -11961.709} C_VEL
LIN {X 0,Y 534.069,Z 835.138,A -85,B 0,C 180,E1 -11962.653,E2 -11962.653} C_VEL
LIN {X 0,Y 533.892,Z 840.894,A -85,B 0,C 180,E1 -11963.597,E2 -11963.597} C_VEL
LIN {X 0,Y 533.751,Z 846.463,A -85,B 0,C 180,E1 -11964.729,E2 -11964.729} C_VEL
LIN {X 0,Y 533.663,Z 849.566,A -85,B 0,C 180,E1 -11965.483,E2 -11965.483} C_VEL
LIN {X 0,Y 533.599,Z 854.067,A -85,B 0,C 180,E1 -11966.99,E2 -11966.99} C_VEL
LIN {X 0,Y 533.593,Z 855.723,A -85,B 0,C 180,E1 -11967.743,E2 -11967.743} C_VEL
LIN {X 0,Y 533.567,Z 857.576,A -85,B 0,C 180,E1 -11969.248,E2 -11969.248} C_VEL
LIN {X 0,Y 533.555,Z 857.888,A -85,B 0,C 180,E1 -11970,E2 -11970} C_VEL
LIN {X 0,Y 533.573,Z 857.291,A -85,B 0,C 180,E1 -11971.505,E2 -11971.505} C_VEL
LIN {X 0,Y 533.602,Z 854.89,A -85,B 0,C 180,E1 -11973.01,E2 -11973.01} C_VEL
LIN {X 0,Y 533.613,Z 852.56,A -85,B 0,C 180,E1 -11973.964,E2 -11973.964} C_VEL
LIN {X 0,Y 533.72,Z 849.579,A -85,B 0,C 180,E1 -11974.894,E2 -11974.894} C_VEL
LIN {X 0,Y 533.875,Z 844.867,A -85,B 0,C 180,E1 -11976.025,E2 -11976.025} C_VEL
LIN {X 0,Y 534.083,Z 838.876,A -85,B 0,C 180,E1 -11977.157,E2 -11977.157} C_VEL
LIN {X 0,Y 534.441,Z 831.365,A -85,B 0,C 180,E1 -11978.289,E2 -11978.289} C_VEL
LIN {X 0,Y 534.875,Z 823.767,A -85,B 0,C 180,E1 -11979.231,E2 -11979.231} C_VEL
LIN {X 0,Y 535.352,Z 815.579,A -85,B 0,C 180,E1 -11980.079,E2 -11980.079} C_VEL
LIN {X 0,Y 535.809,Z 806.897,A -85,B 0,C 180,E1 -11980.832,E2 -11980.832} C_VEL
LIN {X 0,Y 536.263,Z 797.281,A -85,B 0,C 180,E1 -11981.524,E2 -11981.524} C_VEL
LIN {X 0,Y 536.683,Z 788.454,A -85,B 0,C 180,E1 -11982.053,E2 -11982.053} C_VEL
LIN {X 0,Y 537.127,Z 777.751,A -85,B 0,C 180,E1 -11982.569,E2 -11982.569} C_VEL
LIN {X 0,Y 537.544,Z 766.375,A -85,B 0,C 180,E1 -11982.99,E2 -11982.99} C_VEL
LIN {X 0,Y 537.888,Z 754.934,A -85,B 0,C 180,E1 -11983.293,E2 -11983.293} C_VEL
LIN {X 0,Y 538.305,Z 731.359,A -85,B 0,C 180,E1 -11983.689,E2 -11983.689} C_VEL
LIN {X 0,Y 539.145,Z 669.032,A -85,B 0,C 180,E1 -11984.699,E2 -11984.699} C_VEL
LIN {X 0,Y 536.634,Z 651.231,A -85,B 0,C 180,E1 -11985.093,E2 -11985.093} C_VEL
LIN {X 0,Y 535.673,Z 645.772,A -85,B 0,C 180,E1 -11985.233,E2 -11985.233} C_VEL
LIN {X 0,Y 536.706,Z 627.207,A -85,B 0,C 180,E1 -11988.45,E2 -11988.45} C_VEL
LIN {X 0,Y 538.089,Z 608.518,A -85,B 0,C 180,E1 -11991.777,E2 -11991.777} C_VEL
LIN {X 0,Y 537.717,Z 603.998,A -85,B 0,C 180,E1 -11992.642,E2 -11992.642} C_VEL
LIN {X 0,Y 535.742,Z 593.684,A -85,B 0,C 180,E1 -11994.732,E2 -11994.732} C_VEL
LIN {X 0,Y 535.097,Z 590.767,A -85,B 0,C 180,E1 -11995.368,E2 -11995.368} C_VEL
LIN {X 0,Y 535.075,Z 590.773,A -85,B 0,C 180,E1 -11998.116,E2 -11998.116} C_VEL
LIN {X 0,Y 535.075,Z 590.767,A -85,B 0,C 180,E1 -12000.7,E2 -12000.7} C_VEL
LIN {X 0,Y 535.055,Z 590.772,A -85,B 0,C 180,E1 -12003.355,E2 -12003.355} C_VEL
LIN {X 0,Y 535.116,Z 590.759,A -85,B 0,C 180,E1 -12006.089,E2 -12006.089} C_VEL
LIN {X 0,Y 535.046,Z 590.764,A -85,B 0,C 180,E1 -12008.931,E2 -12008.931} C_VEL
LIN {X 0,Y 535.074,Z 590.763,A -85,B 0,C 180,E1 -12011.884,E2 -12011.884} C_VEL
LIN {X 0,Y 535.1,Z 590.764,A -85,B 0,C 180,E1 -12015.02,E2 -12015.02} C_VEL
LIN {X 0,Y 535.098,Z 590.764,A -85,B 0,C 180,E1 -12017.142,E2 -12017.142} C_VEL
LIN {X 0,Y 535.1,Z 590.761,A -85,B 0,C 180,E1 -12020.103,E2 -12020.103} C_VEL
LIN {X 0,Y 535.104,Z 590.764,A -85,B 0,C 180,E1 -12022.986,E2 -12022.986} C_VEL
LIN {X 0,Y 535.116,Z 590.759,A -85,B 0,C 180,E1 -12025.747,E2 -12025.747} C_VEL
LIN {X 0,Y 535.084,Z 590.764,A -85,B 0,C 180,E1 -12028.425,E2 -12028.425} C_VEL
LIN {X 0,Y 535.101,Z 590.763,A -85,B 0,C 180,E1 -12031.286,E2 -12031.286} C_VEL
LIN {X 0,Y 535.086,Z 590.764,A -85,B 0,C 180,E1 -12033.572,E2 -12033.572} C_VEL
LIN {X 0,Y 535.098,Z 590.766,A -85,B 0,C 180,E1 -12036.392,E2 -12036.392} C_VEL
LIN {X 0,Y 535.136,Z 590.761,A -85,B 0,C 180,E1 -12039.304,E2 -12039.304} C_VEL
LIN {X 0,Y 535.101,Z 590.767,A -85,B 0,C 180,E1 -12041.69,E2 -12041.69} C_VEL
LIN {X 0,Y 535.134,Z 590.764,A -85,B 0,C 180,E1 -12044.045,E2 -12044.045} C_VEL
LIN {X 0,Y 535.175,Z 590.758,A -85,B 0,C 180,E1 -12046.374,E2 -12046.374} C_VEL
LIN {X 0,Y 535.198,Z 590.876,A -85,B 0,C 180,E1 -12047.577,E2 -12047.577} C_VEL
LIN {X 0,Y 537.116,Z 600.781,A -85,B 0,C 180,E1 -12049.86,E2 -12049.86} C_VEL
LIN {X 0,Y 537.29,Z 606.079,A -85,B 0,C 180,E1 -12051,E2 -12051} C_VEL
LIN {X 0,Y 536.717,Z 614.238,A -85,B 0,C 180,E1 -12052.678,E2 -12052.678} C_VEL
LIN {X 0,Y 536.036,Z 624.964,A -85,B 0,C 180,E1 -12054.846,E2 -12054.846} C_VEL
LIN {X 0,Y 539.517,Z 643.62,A -85,B 0,C 180,E1 -12055.299,E2 -12055.299} C_VEL
LIN {X 0,Y 538.267,Z 709.927,A -85,B 0,C 180,E1 -12056.363,E2 -12056.363} C_VEL
LIN {X 0,Y 537.865,Z 732.853,A -85,B 0,C 180,E1 -12056.757,E2 -12056.757} C_VEL
LIN {X 0,Y 537.526,Z 745.549,A -85,B 0,C 180,E1 -12057.105,E2 -12057.105} C_VEL
LIN {X 0,Y 537.122,Z 759.245,A -85,B 0,C 180,E1 -12057.664,E2 -12057.664} C_VEL
LIN {X 0,Y 536.788,Z 769.619,A -85,B 0,C 180,E1 -12058.224,E2 -12058.224} C_VEL
LIN {X 0,Y 536.392,Z 779.471,A -85,B 0,C 180,E1 -12058.877,E2 -12058.877} C_VEL
LIN {X 0,Y 535.895,Z 788.772,A -85,B 0,C 180,E1 -12059.625,E2 -12059.625} C_VEL
LIN {X 0,Y 535.425,Z 796.611,A -85,B 0,C 180,E1 -12060.375,E2 -12060.375} C_VEL
LIN {X 0,Y 534.841,Z 804.78,A -85,B 0,C 180,E1 -12061.313,E2 -12061.313} C_VEL
LIN {X 0,Y 534.537,Z 811.557,A -85,B 0,C 180,E1 -12062.253,E2 -12062.253} C_VEL
LIN {X 0,Y 534.168,Z 816.271,A -85,B 0,C 180,E1 -12063.006,E2 -12063.006} C_VEL
LIN {X 0,Y 534.042,Z 822.262,A -85,B 0,C 180,E1 -12064.209,E2 -12064.209} C_VEL
LIN {X 0,Y 533.859,Z 826.463,A -85,B 0,C 180,E1 -12065.269,E2 -12065.269} C_VEL
LIN {X 0,Y 533.765,Z 828.806,A -85,B 0,C 180,E1 -12066.026,E2 -12066.026} C_VEL
LIN {X 0,Y 533.539,Z 832.263,A -85,B 0,C 180,E1 -12067.543,E2 -12067.543} C_VEL
LIN {X 0,Y 533.498,Z 833.838,A -85,B 0,C 180,E1 -12069.064,E2 -12069.064} C_VEL
LIN {X 0,Y 533.539,Z 834.037,A -85,B 0,C 180,E1 -12070.061,E2 -12070.061} C_VEL
LIN {X 0,Y 533.498,Z 833.132,A -85,B 0,C 180,E1 -12071.358,E2 -12071.358} C_VEL
LIN {X 0,Y 533.47,Z 832.096,A -85,B 0,C 180,E1 -12072.127,E2 -12072.127} C_VEL
LIN {X 0,Y 533.62,Z 829.585,A -85,B 0,C 180,E1 -12073.28,E2 -12073.28} C_VEL
LIN {X 0,Y 533.739,Z 825.995,A -85,B 0,C 180,E1 -12074.438,E2 -12074.438} C_VEL
LIN {X 0,Y 533.881,Z 821.202,A -85,B 0,C 180,E1 -12075.602,E2 -12075.602} C_VEL
LIN {X 0,Y 534.092,Z 814.881,A -85,B 0,C 180,E1 -12076.789,E2 -12076.789} C_VEL
LIN {X 0,Y 534.317,Z 808.658,A -85,B 0,C 180,E1 -12077.745,E2 -12077.745} C_VEL
LIN {X 0,Y 534.684,Z 800.941,A -85,B 0,C 180,E1 -12078.72,E2 -12078.72} C_VEL
LIN {X 0,Y 535.051,Z 791.97,A -85,B 0,C 180,E1 -12079.653,E2 -12079.653} C_VEL
LIN {X 0,Y 535.36,Z 783.545,A -85,B 0,C 180,E1 -12080.386,E2 -12080.386} C_VEL
LIN {X 0,Y 535.804,Z 774.077,A -85,B 0,C 180,E1 -12081.069,E2 -12081.069} C_VEL
LIN {X 0,Y 536.165,Z 763.664,A -85,B 0,C 180,E1 -12081.682,E2 -12081.682} C_VEL
LIN {X 0,Y 536.467,Z 753.698,A -85,B 0,C 180,E1 -12082.153,E2 -12082.153} C_VEL
LIN {X 0,Y 536.671,Z 743.034,A -85,B 0,C 180,E1 -12082.544,E2 -12082.544} C_VEL
LIN {X 0,Y 536.929,Z 731.899,A -85,B 0,C 180,E1 -12082.836,E2 -12082.836} C_VEL
LIN {X 0,Y 537.316,Z 711.31,A -85,B 0,C 180,E1 -12083.174,E2 -12083.174} C_VEL
LIN {X 0,Y 538.115,Z 642.945,A -85,B 0,C 180,E1 -12084.217,E2 -12084.217} C_VEL
LIN {X 0,Y 535.347,Z 623.578,A -85,B 0,C 180,E1 -12084.6,E2 -12084.6} C_VEL
LIN {X 0,Y 536.031,Z 607.762,A -85,B 0,C 180,E1 -12087.637,E2 -12087.637} C_VEL
LIN {X 0,Y 536.316,Z 598.001,A -85,B 0,C 180,E1 -12089.539,E2 -12089.539} C_VEL
LIN {X 0,Y 535.185,Z 590.754,A -85,B 0,C 180,E1 -12091.019,E2 -12091.019} C_VEL
LIN {X 0,Y 535.103,Z 590.76,A -85,B 0,C 180,E1 -12094.445,E2 -12094.445} C_VEL
LIN {X 0,Y 535.1,Z 590.758,A -85,B 0,C 180,E1 -12097.023,E2 -12097.023} C_VEL
LIN {X 0,Y 535.097,Z 590.766,A -85,B 0,C 180,E1 -12099.897,E2 -12099.897} C_VEL
LIN {X 0,Y 535.089,Z 590.759,A -85,B 0,C 180,E1 -12102.897,E2 -12102.897} C_VEL
LIN {X 0,Y 535.097,Z 590.758,A -85,B 0,C 180,E1 -12105.02,E2 -12105.02} C_VEL
LIN {X 0,Y 535.087,Z 590.76,A -85,B 0,C 180,E1 -12107.142,E2 -12107.142} C_VEL
LIN {X 0,Y 535.096,Z 590.766,A -85,B 0,C 180,E1 -12110.102,E2 -12110.102} C_VEL
LIN {X 0,Y 535.099,Z 590.758,A -85,B 0,C 180,E1 -12112.985,E2 -12112.985} C_VEL
LIN {X 0,Y 535.11,Z 590.762,A -85,B 0,C 180,E1 -12115.746,E2 -12115.746} C_VEL
LIN {X 0,Y 535.079,Z 590.763,A -85,B 0,C 180,E1 -12118.424,E2 -12118.424} C_VEL
LIN {X 0,Y 535.095,Z 590.759,A -85,B 0,C 180,E1 -12121.286,E2 -12121.286} C_VEL
LIN {X 0,Y 535.09,Z 590.763,A -85,B 0,C 180,E1 -12123.572,E2 -12123.572} C_VEL
LIN {X 0,Y 535.092,Z 590.762,A -85,B 0,C 180,E1 -12126.391,E2 -12126.391} C_VEL
LIN {X 0,Y 535.129,Z 590.755,A -85,B 0,C 180,E1 -12129.304,E2 -12129.304} C_VEL
LIN {X 0,Y 535.11,Z 590.759,A -85,B 0,C 180,E1 -12132.478,E2 -12132.478} C_VEL
LIN {X 0,Y 535.203,Z 590.749,A -85,B 0,C 180,E1 -12135.601,E2 -12135.601} C_VEL
LIN {X 0,Y 535.224,Z 590.743,A -85,B 0,C 180,E1 -12138.965,E2 -12138.965} C_VEL
LIN {X 0,Y 535.249,Z 590.742,A -85,B 0,C 180,E1 -12142.48,E2 -12142.48} C_VEL
LIN {X 0,Y 535.245,Z 590.74,A -85,B 0,C 180,E1 -12143.049,E2 -12143.049} C_VEL
LIN {X 0,Y 534.626,Z 590.823,A -85,B 0,C 180,E1 -12143.677,E2 -12143.677} C_VEL
LIN {X 0,Y 531.857,Z 591.17,A -85,B 0,C 180,E1 -12144.697,E2 -12144.697} C_VEL
LIN {X 0,Y 529.449,Z 591.471,A -85,B 0,C 180,E1 -12145.519,E2 -12145.519} C_VEL
LIN {X 0,Y 528.343,Z 591.606,A -85,B 0,C 180,E1 -12146.152,E2 -12146.152} C_VEL
LIN {X 0,Y 528.216,Z 591.619,A -85,B 0,C 180,E1 -12146.367,E2 -12146.367} C_VEL
LIN {X 0,Y 528.408,Z 591.601,A -85,B 0,C 180,E1 -12150,E2 -12150} C_VEL
LIN {X 0,Y 528.259,Z 591.617,A -85,B 0,C 180,E1 -12153.801,E2 -12153.801} C_VEL
LIN {X 0,Y 528.216,Z 591.616,A -85,B 0,C 180,E1 -12156.854,E2 -12156.854} C_VEL
LIN {X 0,Y 528.133,Z 591.634,A -85,B 0,C 180,E1 -12159.928,E2 -12159.928} C_VEL
LIN {X 0,Y 528.115,Z 591.633,A -85,B 0,C 180,E1 -12162.252,E2 -12162.252} C_VEL
LIN {X 0,Y 528.163,Z 591.623,A -85,B 0,C 180,E1 -12164.594,E2 -12164.594} C_VEL
LIN {X 0,Y 528.069,Z 591.64,A -85,B 0,C 180,E1 -12167.763,E2 -12167.763} C_VEL
LIN {X 0,Y 528.087,Z 591.638,A -85,B 0,C 180,E1 -12170.173,E2 -12170.173} C_VEL
LIN {X 0,Y 528.047,Z 591.638,A -85,B 0,C 180,E1 -12172.624,E2 -12172.624} C_VEL
LIN {X 0,Y 528.031,Z 591.642,A -85,B 0,C 180,E1 -12175.574,E2 -12175.574} C_VEL
LIN {X 0,Y 528.043,Z 591.639,A -85,B 0,C 180,E1 -12178.525,E2 -12178.525} C_VEL
LIN {X 0,Y 528.062,Z 591.635,A -85,B 0,C 180,E1 -12181.152,E2 -12181.152} C_VEL
LIN {X 0,Y 528.054,Z 591.643,A -85,B 0,C 180,E1 -12183.856,E2 -12183.856} C_VEL
LIN {X 0,Y 528.098,Z 591.631,A -85,B 0,C 180,E1 -12186.645,E2 -12186.645} C_VEL
LIN {X 0,Y 528.057,Z 591.64,A -85,B 0,C 180,E1 -12189.706,E2 -12189.706} C_VEL
LIN {X 0,Y 528.05,Z 591.638,A -85,B 0,C 180,E1 -12192.571,E2 -12192.571} C_VEL
LIN {X 0,Y 528.041,Z 591.638,A -85,B 0,C 180,E1 -12195.329,E2 -12195.329} C_VEL
LIN {X 0,Y 528.036,Z 591.64,A -85,B 0,C 180,E1 -12198.452,E2 -12198.452} C_VEL
LIN {X 0,Y 528.048,Z 591.638,A -85,B 0,C 180,E1 -12201.432,E2 -12201.432} C_VEL
LIN {X 0,Y 528.084,Z 591.636,A -85,B 0,C 180,E1 -12204.296,E2 -12204.296} C_VEL
LIN {X 0,Y 528.033,Z 591.638,A -85,B 0,C 180,E1 -12207.053,E2 -12207.053} C_VEL
LIN {X 0,Y 528.053,Z 591.641,A -85,B 0,C 180,E1 -12209.732,E2 -12209.732} C_VEL
LIN {X 0,Y 528.061,Z 591.635,A -85,B 0,C 180,E1 -12212.713,E2 -12212.713} C_VEL
LIN {X 0,Y 528.036,Z 591.643,A -85,B 0,C 180,E1 -12215.719,E2 -12215.719} C_VEL
LIN {X 0,Y 528.079,Z 591.638,A -85,B 0,C 180,E1 -12218.199,E2 -12218.199} C_VEL
LIN {X 0,Y 528.092,Z 591.632,A -85,B 0,C 180,E1 -12220.635,E2 -12220.635} C_VEL
LIN {X 0,Y 528.076,Z 591.64,A -85,B 0,C 180,E1 -12223.827,E2 -12223.827} C_VEL
LIN {X 0,Y 528.135,Z 591.631,A -85,B 0,C 180,E1 -12226.189,E2 -12226.189} C_VEL
LIN {X 0,Y 528.18,Z 591.621,A -85,B 0,C 180,E1 -12229.301,E2 -12229.301} C_VEL
LIN {X 0,Y 528.201,Z 591.621,A -85,B 0,C 180,E1 -12232.38,E2 -12232.38} C_VEL
LIN {X 0,Y 528.241,Z 591.613,A -85,B 0,C 180,E1 -12234.674,E2 -12234.674} C_VEL
LIN {X 0,Y 528.254,Z 591.616,A -85,B 0,C 180,E1 -12236.199,E2 -12236.199} C_VEL
LIN {X 0,Y 528.411,Z 591.6,A -85,B 0,C 180,E1 -12240,E2 -12240} C_VEL
LIN {X 0,Y 528.252,Z 591.618,A -85,B 0,C 180,E1 -12243.802,E2 -12243.802} C_VEL
LIN {X 0,Y 528.222,Z 591.615,A -85,B 0,C 180,E1 -12246.854,E2 -12246.854} C_VEL
LIN {X 0,Y 528.142,Z 591.634,A -85,B 0,C 180,E1 -12249.928,E2 -12249.928} C_VEL
LIN {X 0,Y 528.087,Z 591.636,A -85,B 0,C 180,E1 -12252.253,E2 -12252.253} C_VEL
LIN {X 0,Y 528.126,Z 591.628,A -85,B 0,C 180,E1 -12254.596,E2 -12254.596} C_VEL
LIN {X 0,Y 528.055,Z 591.641,A -85,B 0,C 180,E1 -12257.763,E2 -12257.763} C_VEL
LIN {X 0,Y 528.029,Z 591.645,A -85,B 0,C 180,E1 -12260.176,E2 -12260.176} C_VEL
LIN {X 0,Y 528.036,Z 591.639,A -85,B 0,C 180,E1 -12262.624,E2 -12262.624} C_VEL
LIN {X 0,Y 528.027,Z 591.643,A -85,B 0,C 180,E1 -12265.572,E2 -12265.572} C_VEL
LIN {X 0,Y 528.044,Z 591.639,A -85,B 0,C 180,E1 -12268.525,E2 -12268.525} C_VEL
LIN {X 0,Y 528.02,Z 591.64,A -85,B 0,C 180,E1 -12271.155,E2 -12271.155} C_VEL
LIN {X 0,Y 528.008,Z 591.649,A -85,B 0,C 180,E1 -12273.86,E2 -12273.86} C_VEL
LIN {X 0,Y 528.036,Z 591.639,A -85,B 0,C 180,E1 -12276.65,E2 -12276.65} C_VEL
LIN {X 0,Y 528.029,Z 591.644,A -85,B 0,C 180,E1 -12279.701,E2 -12279.701} C_VEL
LIN {X 0,Y 528.045,Z 591.638,A -85,B 0,C 180,E1 -12282.571,E2 -12282.571} C_VEL
LIN {X 0,Y 528.034,Z 591.644,A -85,B 0,C 180,E1 -12285.751,E2 -12285.751} C_VEL
LIN {X 0,Y 528.017,Z 591.643,A -85,B 0,C 180,E1 -12288.45,E2 -12288.45} C_VEL
LIN {X 0,Y 527.992,Z 591.645,A -85,B 0,C 180,E1 -12291.427,E2 -12291.427} C_VEL
LIN {X 0,Y 528.031,Z 591.643,A -85,B 0,C 180,E1 -12294.291,E2 -12294.291} C_VEL
LIN {X 0,Y 528.009,Z 591.641,A -85,B 0,C 180,E1 -12297.051,E2 -12297.051} C_VEL
LIN {X 0,Y 528.031,Z 591.644,A -85,B 0,C 180,E1 -12299.73,E2 -12299.73} C_VEL
LIN {X 0,Y 528.038,Z 591.638,A -85,B 0,C 180,E1 -12302.717,E2 -12302.717} C_VEL
LIN {X 0,Y 528.092,Z 591.817,A -85,B 0,C 180,E1 -12305.722,E2 -12305.722} C_VEL
LIN {X 0,Y 530.292,Z 604.183,A -85,B 0,C 180,E1 -12307.991,E2 -12307.991} C_VEL
LIN {X 0,Y 529.648,Z 617.495,A -85,B 0,C 180,E1 -12310.292,E2 -12310.292} C_VEL
LIN {X 0,Y 528.644,Z 635.967,A -85,B 0,C 180,E1 -12313.449,E2 -12313.449} C_VEL
LIN {X 0,Y 528.156,Z 646.691,A -85,B 0,C 180,E1 -12315.267,E2 -12315.267} C_VEL
LIN {X 0,Y 531.019,Z 671.01,A -85,B 0,C 180,E1 -12315.725,E2 -12315.725} C_VEL
LIN {X 0,Y 529.948,Z 753.945,A -85,B 0,C 180,E1 -12317.04,E2 -12317.04} C_VEL
LIN {X 0,Y 529.753,Z 763.674,A -85,B 0,C 180,E1 -12317.278,E2 -12317.278} C_VEL
LIN {X 0,Y 529.452,Z 773.02,A -85,B 0,C 180,E1 -12317.586,E2 -12317.586} C_VEL
LIN {X 0,Y 529.122,Z 783.968,A -85,B 0,C 180,E1 -12318.063,E2 -12318.063} C_VEL
LIN {X 0,Y 528.806,Z 794.384,A -85,B 0,C 180,E1 -12318.641,E2 -12318.641} C_VEL
LIN {X 0,Y 528.439,Z 803.015,A -85,B 0,C 180,E1 -12319.222,E2 -12319.222} C_VEL
LIN {X 0,Y 528.004,Z 812.277,A -85,B 0,C 180,E1 -12319.973,E2 -12319.973} C_VEL
LIN {X 0,Y 527.571,Z 821.054,A -85,B 0,C 180,E1 -12320.833,E2 -12320.833} C_VEL
LIN {X 0,Y 527.26,Z 827.693,A -85,B 0,C 180,E1 -12321.597,E2 -12321.597} C_VEL
LIN {X 0,Y 526.997,Z 834.663,A -85,B 0,C 180,E1 -12322.554,E2 -12322.554} C_VEL
LIN {X 0,Y 526.811,Z 840.481,A -85,B 0,C 180,E1 -12323.511,E2 -12323.511} C_VEL
LIN {X 0,Y 526.657,Z 846.105,A -85,B 0,C 180,E1 -12324.658,E2 -12324.658} C_VEL
LIN {X 0,Y 526.558,Z 850.507,A -85,B 0,C 180,E1 -12325.805,E2 -12325.805} C_VEL
LIN {X 0,Y 526.506,Z 853.803,A -85,B 0,C 180,E1 -12326.95,E2 -12326.95} C_VEL
LIN {X 0,Y 526.508,Z 855.459,A -85,B 0,C 180,E1 -12327.713,E2 -12327.713} C_VEL
LIN {X 0,Y 526.491,Z 857.393,A -85,B 0,C 180,E1 -12329.238,E2 -12329.238} C_VEL
LIN {X 0,Y 526.478,Z 857.704,A -85,B 0,C 180,E1 -12330,E2 -12330} C_VEL
LIN {X 0,Y 526.481,Z 857.17,A -85,B 0,C 180,E1 -12331.525,E2 -12331.525} C_VEL
LIN {X 0,Y 526.509,Z 854.807,A -85,B 0,C 180,E1 -12333.051,E2 -12333.051} C_VEL
LIN {X 0,Y 526.551,Z 851.948,A -85,B 0,C 180,E1 -12334.195,E2 -12334.195} C_VEL
LIN {X 0,Y 526.665,Z 848.02,A -85,B 0,C 180,E1 -12335.342,E2 -12335.342} C_VEL
LIN {X 0,Y 526.8,Z 844.849,A -85,B 0,C 180,E1 -12336.106,E2 -12336.106} C_VEL
LIN {X 0,Y 527.105,Z 837.703,A -85,B 0,C 180,E1 -12337.445,E2 -12337.445} C_VEL
LIN {X 0,Y 527.398,Z 831.42,A -85,B 0,C 180,E1 -12338.401,E2 -12338.401} C_VEL
LIN {X 0,Y 527.846,Z 823.851,A -85,B 0,C 180,E1 -12339.355,E2 -12339.355} C_VEL
LIN {X 0,Y 528.348,Z 815.705,A -85,B 0,C 180,E1 -12340.214,E2 -12340.214} C_VEL
LIN {X 0,Y 528.849,Z 807.119,A -85,B 0,C 180,E1 -12340.976,E2 -12340.976} C_VEL
LIN {X 0,Y 529.353,Z 797.059,A -85,B 0,C 180,E1 -12341.714,E2 -12341.714} C_VEL
LIN {X 0,Y 529.855,Z 787.143,A -85,B 0,C 180,E1 -12342.308,E2 -12342.308} C_VEL
LIN {X 0,Y 530.297,Z 777.375,A -85,B 0,C 180,E1 -12342.782,E2 -12342.782} C_VEL
LIN {X 0,Y 530.691,Z 766.752,A -85,B 0,C 180,E1 -12343.185,E2 -12343.185} C_VEL
LIN {X 0,Y 531.071,Z 755.607,A -85,B 0,C 180,E1 -12343.491,E2 -12343.491} C_VEL
LIN {X 0,Y 531.454,Z 735.342,A -85,B 0,C 180,E1 -12343.845,E2 -12343.845} C_VEL
LIN {X 0,Y 532.492,Z 670.54,A -85,B 0,C 180,E1 -12344.911,E2 -12344.911} C_VEL
LIN {X 0,Y 530.222,Z 653.865,A -85,B 0,C 180,E1 -12345.29,E2 -12345.29} C_VEL
LIN {X 0,Y 528.717,Z 645.537,A -85,B 0,C 180,E1 -12345.512,E2 -12345.512} C_VEL
LIN {X 0,Y 529.925,Z 626.353,A -85,B 0,C 180,E1 -12348.895,E2 -12348.895} C_VEL
LIN {X 0,Y 531.186,Z 609.973,A -85,B 0,C 180,E1 -12351.871,E2 -12351.871} C_VEL
LIN {X 0,Y 530.971,Z 606.355,A -85,B 0,C 180,E1 -12352.568,E2 -12352.568} C_VEL
LIN {X 0,Y 528.606,Z 594.197,A -85,B 0,C 180,E1 -12355.089,E2 -12355.089} C_VEL
LIN {X 0,Y 528.031,Z 591.648,A -85,B 0,C 180,E1 -12355.654,E2 -12355.654} C_VEL
LIN {X 0,Y 528.037,Z 591.649,A -85,B 0,C 180,E1 -12358.525,E2 -12358.525} C_VEL
LIN {X 0,Y 528.021,Z 591.648,A -85,B 0,C 180,E1 -12361.155,E2 -12361.155} C_VEL
LIN {X 0,Y 528.015,Z 591.648,A -85,B 0,C 180,E1 -12363.86,E2 -12363.86} C_VEL
LIN {X 0,Y 528.073,Z 591.634,A -85,B 0,C 180,E1 -12366.648,E2 -12366.648} C_VEL
LIN {X 0,Y 528.037,Z 591.638,A -85,B 0,C 180,E1 -12369.702,E2 -12369.702} C_VEL
LIN {X 0,Y 528.048,Z 591.637,A -85,B 0,C 180,E1 -12372.571,E2 -12372.571} C_VEL
LIN {X 0,Y 528.058,Z 591.641,A -85,B 0,C 180,E1 -12375.749,E2 -12375.749} C_VEL
LIN {X 0,Y 528.044,Z 591.641,A -85,B 0,C 180,E1 -12378.452,E2 -12378.452} C_VEL
LIN {X 0,Y 528.029,Z 591.643,A -85,B 0,C 180,E1 -12380.451,E2 -12380.451} C_VEL
LIN {X 0,Y 528.078,Z 591.64,A -85,B 0,C 180,E1 -12383.353,E2 -12383.353} C_VEL
LIN {X 0,Y 528.051,Z 591.639,A -85,B 0,C 180,E1 -12386.143,E2 -12386.143} C_VEL
LIN {X 0,Y 528.058,Z 591.644,A -85,B 0,C 180,E1 -12388.847,E2 -12388.847} C_VEL
LIN {X 0,Y 528.048,Z 591.641,A -85,B 0,C 180,E1 -12391.476,E2 -12391.476} C_VEL
LIN {X 0,Y 528.038,Z 591.645,A -85,B 0,C 180,E1 -12394.426,E2 -12394.426} C_VEL
LIN {X 0,Y 528.048,Z 591.644,A -85,B 0,C 180,E1 -12397.376,E2 -12397.376} C_VEL
LIN {X 0,Y 528.094,Z 591.644,A -85,B 0,C 180,E1 -12400.343,E2 -12400.343} C_VEL
LIN {X 0,Y 528.093,Z 591.639,A -85,B 0,C 180,E1 -12403.034,E2 -12403.034} C_VEL
LIN {X 0,Y 528.139,Z 591.633,A -85,B 0,C 180,E1 -12406.189,E2 -12406.189} C_VEL
LIN {X 0,Y 528.101,Z 591.65,A -85,B 0,C 180,E1 -12407.261,E2 -12407.261} C_VEL
LIN {X 0,Y 530.171,Z 602.078,A -85,B 0,C 180,E1 -12409.726,E2 -12409.726} C_VEL
LIN {X 0,Y 530.407,Z 607.327,A -85,B 0,C 180,E1 -12410.882,E2 -12410.882} C_VEL
LIN {X 0,Y 529.544,Z 620.108,A -85,B 0,C 180,E1 -12413.544,E2 -12413.544} C_VEL
LIN {X 0,Y 529.133,Z 625.097,A -85,B 0,C 180,E1 -12414.564,E2 -12414.564} C_VEL
LIN {X 0,Y 532.644,Z 643.747,A -85,B 0,C 180,E1 -12415.049,E2 -12415.049} C_VEL
LIN {X 0,Y 532.795,Z 648.965,A -85,B 0,C 180,E1 -12415.145,E2 -12415.145} C_VEL
LIN {X 0,Y 531.096,Z 731.135,A -85,B 0,C 180,E1 -12416.503,E2 -12416.503} C_VEL
LIN {X 0,Y 530.838,Z 741.329,A -85,B 0,C 180,E1 -12416.761,E2 -12416.761} C_VEL
LIN {X 0,Y 530.565,Z 750.297,A -85,B 0,C 180,E1 -12417.067,E2 -12417.067} C_VEL
LIN {X 0,Y 530.227,Z 760.915,A -85,B 0,C 180,E1 -12417.539,E2 -12417.539} C_VEL
LIN {X 0,Y 529.853,Z 771.015,A -85,B 0,C 180,E1 -12418.106,E2 -12418.106} C_VEL
LIN {X 0,Y 529.436,Z 780.622,A -85,B 0,C 180,E1 -12418.768,E2 -12418.768} C_VEL
LIN {X 0,Y 528.996,Z 788.716,A -85,B 0,C 180,E1 -12419.431,E2 -12419.431} C_VEL
LIN {X 0,Y 528.473,Z 796.579,A -85,B 0,C 180,E1 -12420.19,E2 -12420.19} C_VEL
LIN {X 0,Y 527.861,Z 804.764,A -85,B 0,C 180,E1 -12421.14,E2 -12421.14} C_VEL
LIN {X 0,Y 527.527,Z 811.577,A -85,B 0,C 180,E1 -12422.092,E2 -12422.092} C_VEL
LIN {X 0,Y 527.086,Z 817.306,A -85,B 0,C 180,E1 -12423.047,E2 -12423.047} C_VEL
LIN {X 0,Y 526.987,Z 822.695,A -85,B 0,C 180,E1 -12424.162,E2 -12424.162} C_VEL
LIN {X 0,Y 526.766,Z 827.155,A -85,B 0,C 180,E1 -12425.341,E2 -12425.341} C_VEL
LIN {X 0,Y 526.683,Z 829.503,A -85,B 0,C 180,E1 -12426.107,E2 -12426.107} C_VEL
LIN {X 0,Y 526.436,Z 832.655,A -85,B 0,C 180,E1 -12427.646,E2 -12427.646} C_VEL
LIN {X 0,Y 526.423,Z 833.631,A -85,B 0,C 180,E1 -12428.416,E2 -12428.416} C_VEL
LIN {X 0,Y 526.446,Z 834.178,A -85,B 0,C 180,E1 -12430.073,E2 -12430.073} C_VEL
LIN {X 0,Y 526.422,Z 833.871,A -85,B 0,C 180,E1 -12430.735,E2 -12430.735} C_VEL
LIN {X 0,Y 526.388,Z 831.918,A -85,B 0,C 180,E1 -12432.292,E2 -12432.292} C_VEL
LIN {X 0,Y 526.559,Z 829.278,A -85,B 0,C 180,E1 -12433.448,E2 -12433.448} C_VEL
LIN {X 0,Y 526.66,Z 825.44,A -85,B 0,C 180,E1 -12434.637,E2 -12434.637} C_VEL
LIN {X 0,Y 526.846,Z 820.401,A -85,B 0,C 180,E1 -12435.816,E2 -12435.816} C_VEL
LIN {X 0,Y 527.083,Z 813.952,A -85,B 0,C 180,E1 -12436.999,E2 -12436.999} C_VEL
LIN {X 0,Y 527.326,Z 807.34,A -85,B 0,C 180,E1 -12437.988,E2 -12437.988} C_VEL
LIN {X 0,Y 527.635,Z 801.113,A -85,B 0,C 180,E1 -12438.779,E2 -12438.779} C_VEL
LIN {X 0,Y 527.995,Z 792.022,A -85,B 0,C 180,E1 -12439.735,E2 -12439.735} C_VEL
LIN {X 0,Y 528.303,Z 783.697,A -85,B 0,C 180,E1 -12440.468,E2 -12440.468} C_VEL
LIN {X 0,Y 528.766,Z 774.228,A -85,B 0,C 180,E1 -12441.16,E2 -12441.16} C_VEL
LIN {X 0,Y 529.116,Z 764.284,A -85,B 0,C 180,E1 -12441.756,E2 -12441.756} C_VEL
LIN {X 0,Y 529.462,Z 754.623,A -85,B 0,C 180,E1 -12442.226,E2 -12442.226} C_VEL
LIN {X 0,Y 529.65,Z 743.192,A -85,B 0,C 180,E1 -12442.654,E2 -12442.654} C_VEL
LIN {X 0,Y 529.911,Z 732.113,A -85,B 0,C 180,E1 -12442.95,E2 -12442.95} C_VEL
LIN {X 0,Y 530.315,Z 711.74,A -85,B 0,C 180,E1 -12443.292,E2 -12443.292} C_VEL
LIN {X 0,Y 531.093,Z 642.653,A -85,B 0,C 180,E1 -12444.377,E2 -12444.377} C_VEL
LIN {X 0,Y 528.294,Z 623.726,A -85,B 0,C 180,E1 -12444.754,E2 -12444.754} C_VEL
LIN {X 0,Y 529.033,Z 607.958,A -85,B 0,C 180,E1 -12447.821,E2 -12447.821} C_VEL
LIN {X 0,Y 529.315,Z 599.27,A -85,B 0,C 180,E1 -12449.533,E2 -12449.533} C_VEL
LIN {X 0,Y 528.125,Z 591.635,A -85,B 0,C 180,E1 -12451.148,E2 -12451.148} C_VEL
LIN {X 0,Y 528.052,Z 591.643,A -85,B 0,C 180,E1 -12453.856,E2 -12453.856} C_VEL
LIN {X 0,Y 528.075,Z 591.634,A -85,B 0,C 180,E1 -12456.647,E2 -12456.647} C_VEL
LIN {X 0,Y 528.055,Z 591.641,A -85,B 0,C 180,E1 -12459.704,E2 -12459.704} C_VEL
LIN {X 0,Y 528.052,Z 591.637,A -85,B 0,C 180,E1 -12462.57,E2 -12462.57} C_VEL
LIN {X 0,Y 528.043,Z 591.638,A -85,B 0,C 180,E1 -12465.328,E2 -12465.328} C_VEL
LIN {X 0,Y 528.037,Z 591.64,A -85,B 0,C 180,E1 -12468.451,E2 -12468.451} C_VEL
LIN {X 0,Y 528.024,Z 591.642,A -85,B 0,C 180,E1 -12470.451,E2 -12470.451} C_VEL
LIN {X 0,Y 528.074,Z 591.635,A -85,B 0,C 180,E1 -12473.353,E2 -12473.353} C_VEL
LIN {X 0,Y 528.045,Z 591.643,A -85,B 0,C 180,E1 -12476.143,E2 -12476.143} C_VEL
LIN {X 0,Y 528.032,Z 591.639,A -85,B 0,C 180,E1 -12478.846,E2 -12478.846} C_VEL
LIN {X 0,Y 528.042,Z 591.639,A -85,B 0,C 180,E1 -12481.475,E2 -12481.475} C_VEL
LIN {X 0,Y 528.033,Z 591.641,A -85,B 0,C 180,E1 -12484.425,E2 -12484.425} C_VEL
LIN {X 0,Y 528.047,Z 591.638,A -85,B 0,C 180,E1 -12487.376,E2 -12487.376} C_VEL
LIN {X 0,Y 528.088,Z 591.635,A -85,B 0,C 180,E1 -12490.342,E2 -12490.342} C_VEL
LIN {X 0,Y 528.103,Z 591.63,A -85,B 0,C 180,E1 -12493.034,E2 -12493.034} C_VEL
LIN {X 0,Y 528.145,Z 591.63,A -85,B 0,C 180,E1 -12496.189,E2 -12496.189} C_VEL
LIN {X 0,Y 528.175,Z 591.622,A -85,B 0,C 180,E1 -12499.3,E2 -12499.3} C_VEL
LIN {X 0,Y 528.196,Z 591.621,A -85,B 0,C 180,E1 -12502.379,E2 -12502.379} C_VEL
LIN {X 0,Y 528.249,Z 591.612,A -85,B 0,C 180,E1 -12504.674,E2 -12504.674} C_VEL
LIN {X 0,Y 528.216,Z 591.619,A -85,B 0,C 180,E1 -12506.367,E2 -12506.367} C_VEL
LIN {X 0,Y 527.459,Z 591.712,A -85,B 0,C 180,E1 -12507.003,E2 -12507.003} C_VEL
LIN {X 0,Y 524.63,Z 592.071,A -85,B 0,C 180,E1 -12508.037,E2 -12508.037} C_VEL
LIN {X 0,Y 522.329,Z 592.352,A -85,B 0,C 180,E1 -12508.87,E2 -12508.87} C_VEL
LIN {X 0,Y 521.386,Z 592.469,A -85,B 0,C 180,E1 -12509.512,E2 -12509.512} C_VEL
LIN {X 0,Y 521.329,Z 592.478,A -85,B 0,C 180,E1 -12509.729,E2 -12509.729} C_VEL
LIN {X 0,Y 521.155,Z 592.498,A -85,B 0,C 180,E1 -12511.54,E2 -12511.54} C_VEL
LIN {X 0,Y 521.253,Z 592.484,A -85,B 0,C 180,E1 -12514.624,E2 -12514.624} C_VEL
LIN {X 0,Y 521.178,Z 592.492,A -85,B 0,C 180,E1 -12516.947,E2 -12516.947} C_VEL
LIN {X 0,Y 521.114,Z 592.508,A -85,B 0,C 180,E1 -12520.063,E2 -12520.063} C_VEL
LIN {X 0,Y 521.078,Z 592.508,A -85,B 0,C 180,E1 -12522.42,E2 -12522.42} C_VEL
LIN {X 0,Y 521.101,Z 592.502,A -85,B 0,C 180,E1 -12524.797,E2 -12524.797} C_VEL
LIN {X 0,Y 521.009,Z 592.522,A -85,B 0,C 180,E1 -12528.012,E2 -12528.012} C_VEL
LIN {X 0,Y 521.031,Z 592.513,A -85,B 0,C 180,E1 -12530.458,E2 -12530.458} C_VEL
LIN {X 0,Y 520.995,Z 592.515,A -85,B 0,C 180,E1 -12532.947,E2 -12532.947} C_VEL
LIN {X 0,Y 520.988,Z 592.521,A -85,B 0,C 180,E1 -12535.74,E2 -12535.74} C_VEL
LIN {X 0,Y 520.982,Z 592.524,A -85,B 0,C 180,E1 -12538.071,E2 -12538.071} C_VEL
LIN {X 0,Y 521.036,Z 592.51,A -85,B 0,C 180,E1 -12540.72,E2 -12540.72} C_VEL
LIN {X 0,Y 521.04,Z 592.512,A -85,B 0,C 180,E1 -12543.543,E2 -12543.543} C_VEL
LIN {X 0,Y 521.06,Z 592.512,A -85,B 0,C 180,E1 -12546.262,E2 -12546.262} C_VEL
LIN {X 0,Y 520.995,Z 592.516,A -85,B 0,C 180,E1 -12549.189,E2 -12549.189} C_VEL
LIN {X 0,Y 521.009,Z 592.518,A -85,B 0,C 180,E1 -12552.237,E2 -12552.237} C_VEL
LIN {X 0,Y 520.996,Z 592.517,A -85,B 0,C 180,E1 -12555.443,E2 -12555.443} C_VEL
LIN {X 0,Y 521.018,Z 592.512,A -85,B 0,C 180,E1 -12558.838,E2 -12558.838} C_VEL
LIN {X 0,Y 521.017,Z 592.519,A -85,B 0,C 180,E1 -12561.8,E2 -12561.8} C_VEL
LIN {X 0,Y 521.009,Z 592.514,A -85,B 0,C 180,E1 -12564.684,E2 -12564.684} C_VEL
LIN {X 0,Y 520.972,Z 592.52,A -85,B 0,C 180,E1 -12567.467,E2 -12567.467} C_VEL
LIN {X 0,Y 521.023,Z 592.518,A -85,B 0,C 180,E1 -12570.171,E2 -12570.171} C_VEL
LIN {X 0,Y 521.022,Z 592.512,A -85,B 0,C 180,E1 -12572.801,E2 -12572.801} C_VEL
LIN {X 0,Y 521.022,Z 592.519,A -85,B 0,C 180,E1 -12576.088,E2 -12576.088} C_VEL
LIN {X 0,Y 521.02,Z 592.513,A -85,B 0,C 180,E1 -12578.717,E2 -12578.717} C_VEL
LIN {X 0,Y 521.006,Z 592.514,A -85,B 0,C 180,E1 -12581.177,E2 -12581.177} C_VEL
LIN {X 0,Y 521.024,Z 592.515,A -85,B 0,C 180,E1 -12583.602,E2 -12583.602} C_VEL
LIN {X 0,Y 521.092,Z 592.512,A -85,B 0,C 180,E1 -12585.998,E2 -12585.998} C_VEL
LIN {X 0,Y 521.135,Z 592.498,A -85,B 0,C 180,E1 -12589.154,E2 -12589.154} C_VEL
LIN {X 0,Y 521.165,Z 592.498,A -85,B 0,C 180,E1 -12592.276,E2 -12592.276} C_VEL
LIN {X 0,Y 521.199,Z 592.491,A -85,B 0,C 180,E1 -12594.602,E2 -12594.602} C_VEL
LIN {X 0,Y 521.22,Z 592.493,A -85,B 0,C 180,E1 -12596.148,E2 -12596.148} C_VEL
LIN {X 0,Y 521.365,Z 592.478,A -85,B 0,C 180,E1 -12600,E2 -12600} C_VEL
LIN {X 0,Y 521.243,Z 592.485,A -85,B 0,C 180,E1 -12604.625,E2 -12604.625} C_VEL
LIN {X 0,Y 521.183,Z 592.492,A -85,B 0,C 180,E1 -12606.947,E2 -12606.947} C_VEL
LIN {X 0,Y 521.122,Z 592.507,A -85,B 0,C 180,E1 -12610.063,E2 -12610.063} C_VEL
LIN {X 0,Y 521.053,Z 592.511,A -85,B 0,C 180,E1 -12612.421,E2 -12612.421} C_VEL
LIN {X 0,Y 521.081,Z 592.505,A -85,B 0,C 180,E1 -12614.797,E2 -12614.797} C_VEL
LIN {X 0,Y 520.997,Z 592.523,A -85,B 0,C 180,E1 -12618.012,E2 -12618.012} C_VEL
LIN {X 0,Y 520.987,Z 592.518,A -85,B 0,C 180,E1 -12620.46,E2 -12620.46} C_VEL
LIN {X 0,Y 520.99,Z 592.516,A -85,B 0,C 180,E1 -12622.948,E2 -12622.948} C_VEL
LIN {X 0,Y 520.986,Z 592.522,A -85,B 0,C 180,E1 -12625.738,E2 -12625.738} C_VEL
LIN {X 0,Y 520.983,Z 592.524,A -85,B 0,C 180,E1 -12628.071,E2 -12628.071} C_VEL
LIN {X 0,Y 520.986,Z 592.517,A -85,B 0,C 180,E1 -12630.723,E2 -12630.723} C_VEL
LIN {X 0,Y 520.973,Z 592.521,A -85,B 0,C 180,E1 -12633.531,E2 -12633.531} C_VEL
LIN {X 0,Y 520.996,Z 592.519,A -85,B 0,C 180,E1 -12636.267,E2 -12636.267} C_VEL
LIN {X 0,Y 520.94,Z 592.522,A -85,B 0,C 180,E1 -12638.753,E2 -12638.753} C_VEL
LIN {X 0,Y 520.974,Z 592.518,A -85,B 0,C 180,E1 -12641.208,E2 -12641.208} C_VEL
LIN {X 0,Y 520.987,Z 592.52,A -85,B 0,C 180,E1 -12644.356,E2 -12644.356} C_VEL
LIN {X 0,Y 520.986,Z 592.517,A -85,B 0,C 180,E1 -12646.711,E2 -12646.711} C_VEL
LIN {X 0,Y 520.96,Z 592.526,A -85,B 0,C 180,E1 -12649.806,E2 -12649.806} C_VEL
LIN {X 0,Y 520.982,Z 592.517,A -85,B 0,C 180,E1 -12652.77,E2 -12652.77} C_VEL
LIN {X 0,Y 520.959,Z 592.523,A -85,B 0,C 180,E1 -12655.619,E2 -12655.619} C_VEL
LIN {X 0,Y 520.956,Z 592.523,A -85,B 0,C 180,E1 -12658.374,E2 -12658.374} C_VEL
LIN {X 0,Y 521.01,Z 592.513,A -85,B 0,C 180,E1 -12661.054,E2 -12661.054} C_VEL
LIN {X 0,Y 520.997,Z 592.519,A -85,B 0,C 180,E1 -12663.662,E2 -12663.662} C_VEL
LIN {X 0,Y 521.05,Z 592.642,A -85,B 0,C 180,E1 -12665.594,E2 -12665.594} C_VEL
LIN {X 0,Y 523.308,Z 605.518,A -85,B 0,C 180,E1 -12667.99,E2 -12667.99} C_VEL
LIN {X 0,Y 522.637,Z 618.362,A -85,B 0,C 180,E1 -12670.239,E2 -12670.239} C_VEL
LIN {X 0,Y 521.606,Z 636.742,A -85,B 0,C 180,E1 -12673.42,E2 -12673.42} C_VEL
LIN {X 0,Y 521.119,Z 646.588,A -85,B 0,C 180,E1 -12675.111,E2 -12675.111} C_VEL
LIN {X 0,Y 524.054,Z 671.753,A -85,B 0,C 180,E1 -12675.595,E2 -12675.595} C_VEL
LIN {X 0,Y 522.933,Z 753.359,A -85,B 0,C 180,E1 -12676.912,E2 -12676.912} C_VEL
LIN {X 0,Y 522.73,Z 763.205,A -85,B 0,C 180,E1 -12677.153,E2 -12677.153} C_VEL
LIN {X 0,Y 522.419,Z 773.812,A -85,B 0,C 180,E1 -12677.514,E2 -12677.514} C_VEL
LIN {X 0,Y 522.157,Z 782.692,A -85,B 0,C 180,E1 -12677.901,E2 -12677.901} C_VEL
LIN {X 0,Y 521.852,Z 791.74,A -85,B 0,C 180,E1 -12678.385,E2 -12678.385} C_VEL
LIN {X 0,Y 521.377,Z 803.185,A -85,B 0,C 180,E1 -12679.159,E2 -12679.159} C_VEL
LIN {X 0,Y 520.97,Z 811.496,A -85,B 0,C 180,E1 -12679.836,E2 -12679.836} C_VEL
LIN {X 0,Y 520.529,Z 820.38,A -85,B 0,C 180,E1 -12680.708,E2 -12680.708} C_VEL
LIN {X 0,Y 520.21,Z 827.109,A -85,B 0,C 180,E1 -12681.483,E2 -12681.483} C_VEL
LIN {X 0,Y 519.939,Z 834.157,A -85,B 0,C 180,E1 -12682.453,E2 -12682.453} C_VEL
LIN {X 0,Y 519.751,Z 840.044,A -85,B 0,C 180,E1 -12683.422,E2 -12683.422} C_VEL
LIN {X 0,Y 519.573,Z 845.729,A -85,B 0,C 180,E1 -12684.585,E2 -12684.585} C_VEL
LIN {X 0,Y 519.464,Z 850.185,A -85,B 0,C 180,E1 -12685.747,E2 -12685.747} C_VEL
LIN {X 0,Y 519.415,Z 853.533,A -85,B 0,C 180,E1 -12686.908,E2 -12686.908} C_VEL
LIN {X 0,Y 519.425,Z 855.192,A -85,B 0,C 180,E1 -12687.682,E2 -12687.682} C_VEL
LIN {X 0,Y 519.418,Z 857.21,A -85,B 0,C 180,E1 -12689.227,E2 -12689.227} C_VEL
LIN {X 0,Y 519.404,Z 857.521,A -85,B 0,C 180,E1 -12690,E2 -12690} C_VEL
LIN {X 0,Y 519.392,Z 857.044,A -85,B 0,C 180,E1 -12691.546,E2 -12691.546} C_VEL
LIN {X 0,Y 519.42,Z 854.725,A -85,B 0,C 180,E1 -12693.092,E2 -12693.092} C_VEL
LIN {X 0,Y 519.461,Z 851.893,A -85,B 0,C 180,E1 -12694.253,E2 -12694.253} C_VEL
LIN {X 0,Y 519.584,Z 847.99,A -85,B 0,C 180,E1 -12695.415,E2 -12695.415} C_VEL
LIN {X 0,Y 519.808,Z 842.915,A -85,B 0,C 180,E1 -12696.577,E2 -12696.577} C_VEL
LIN {X 0,Y 520.047,Z 837.739,A -85,B 0,C 180,E1 -12697.546,E2 -12697.546} C_VEL
LIN {X 0,Y 520.362,Z 831.52,A -85,B 0,C 180,E1 -12698.515,E2 -12698.515} C_VEL
LIN {X 0,Y 520.841,Z 824.031,A -85,B 0,C 180,E1 -12699.482,E2 -12699.482} C_VEL
LIN {X 0,Y 521.432,Z 814.95,A -85,B 0,C 180,E1 -12700.448,E2 -12700.448} C_VEL
LIN {X 0,Y 521.999,Z 806.238,A -85,B 0,C 180,E1 -12701.22,E2 -12701.22} C_VEL
LIN {X 0,Y 522.444,Z 797.143,A -85,B 0,C 180,E1 -12701.896,E2 -12701.896} C_VEL
LIN {X 0,Y 522.943,Z 787.744,A -85,B 0,C 180,E1 -12702.473,E2 -12702.473} C_VEL
LIN {X 0,Y 523.435,Z 777.018,A -85,B 0,C 180,E1 -12703.002,E2 -12703.002} C_VEL
LIN {X 0,Y 523.899,Z 766.337,A -85,B 0,C 180,E1 -12703.408,E2 -12703.408} C_VEL
LIN {X 0,Y 524.289,Z 755.111,A -85,B 0,C 180,E1 -12703.718,E2 -12703.718} C_VEL
LIN {X 0,Y 524.747,Z 732.021,A -85,B 0,C 180,E1 -12704.124,E2 -12704.124} C_VEL
LIN {X 0,Y 525.728,Z 670.946,A -85,B 0,C 180,E1 -12705.157,E2 -12705.157} C_VEL
LIN {X 0,Y 523.619,Z 655.275,A -85,B 0,C 180,E1 -12705.527,E2 -12705.527} C_VEL
LIN {X 0,Y 521.798,Z 645.47,A -85,B 0,C 180,E1 -12705.781,E2 -12705.781} C_VEL
LIN {X 0,Y 523.082,Z 626.665,A -85,B 0,C 180,E1 -12709.152,E2 -12709.152} C_VEL
LIN {X 0,Y 524.286,Z 611.43,A -85,B 0,C 180,E1 -12711.968,E2 -12711.968} C_VEL
LIN {X 0,Y 523.925,Z 607.19,A -85,B 0,C 180,E1 -12712.812,E2 -12712.812} C_VEL
LIN {X 0,Y 521.965,Z 596.803,A -85,B 0,C 180,E1 -12715.006,E2 -12715.006} C_VEL
LIN {X 0,Y 521.01,Z 592.524,A -85,B 0,C 180,E1 -12715.997,E2 -12715.997} C_VEL
LIN {X 0,Y 521.009,Z 592.523,A -85,B 0,C 180,E1 -12719.09,E2 -12719.09} C_VEL
LIN {X 0,Y 520.952,Z 592.528,A -85,B 0,C 180,E1 -12722.106,E2 -12722.106} C_VEL
LIN {X 0,Y 520.979,Z 592.521,A -85,B 0,C 180,E1 -12724.902,E2 -12724.902} C_VEL
LIN {X 0,Y 521.02,Z 592.515,A -85,B 0,C 180,E1 -12727.516,E2 -12727.516} C_VEL
LIN {X 0,Y 520.964,Z 592.518,A -85,B 0,C 180,E1 -12730.193,E2 -12730.193} C_VEL
LIN {X 0,Y 520.989,Z 592.519,A -85,B 0,C 180,E1 -12733.289,E2 -12733.289} C_VEL
LIN {X 0,Y 521.002,Z 592.519,A -85,B 0,C 180,E1 -12736.551,E2 -12736.551} C_VEL
LIN {X 0,Y 521.024,Z 592.518,A -85,B 0,C 180,E1 -12738.838,E2 -12738.838} C_VEL
LIN {X 0,Y 520.954,Z 592.527,A -85,B 0,C 180,E1 -12741.246,E2 -12741.246} C_VEL
LIN {X 0,Y 521.063,Z 592.51,A -85,B 0,C 180,E1 -12743.761,E2 -12743.761} C_VEL
LIN {X 0,Y 521.015,Z 592.517,A -85,B 0,C 180,E1 -12746.551,E2 -12746.551} C_VEL
LIN {X 0,Y 521.021,Z 592.515,A -85,B 0,C 180,E1 -12749.362,E2 -12749.362} C_VEL
LIN {X 0,Y 520.986,Z 592.52,A -85,B 0,C 180,E1 -12751.929,E2 -12751.929} C_VEL
LIN {X 0,Y 520.995,Z 592.522,A -85,B 0,C 180,E1 -12754.518,E2 -12754.518} C_VEL
LIN {X 0,Y 520.998,Z 592.523,A -85,B 0,C 180,E1 -12757.053,E2 -12757.053} C_VEL
LIN {X 0,Y 521.036,Z 592.517,A -85,B 0,C 180,E1 -12759.542,E2 -12759.542} C_VEL
LIN {X 0,Y 521.033,Z 592.522,A -85,B 0,C 180,E1 -12762.797,E2 -12762.797} C_VEL
LIN {X 0,Y 521.096,Z 592.509,A -85,B 0,C 180,E1 -12765.998,E2 -12765.998} C_VEL
LIN {X 0,Y 521.107,Z 592.629,A -85,B 0,C 180,E1 -12766.988,E2 -12766.988} C_VEL
LIN {X 0,Y 523.225,Z 603.394,A -85,B 0,C 180,E1 -12769.588,E2 -12769.588} C_VEL
LIN {X 0,Y 523.512,Z 608.627,A -85,B 0,C 180,E1 -12770.761,E2 -12770.761} C_VEL
LIN {X 0,Y 522.695,Z 619.515,A -85,B 0,C 180,E1 -12773.073,E2 -12773.073} C_VEL
LIN {X 0,Y 522.274,Z 625.61,A -85,B 0,C 180,E1 -12774.299,E2 -12774.299} C_VEL
LIN {X 0,Y 525.783,Z 643.319,A -85,B 0,C 180,E1 -12774.769,E2 -12774.769} C_VEL
LIN {X 0,Y 526.201,Z 646.56,A -85,B 0,C 180,E1 -12774.845,E2 -12774.845} C_VEL
LIN {X 0,Y 524.315,Z 731.654,A -85,B 0,C 180,E1 -12776.29,E2 -12776.29} C_VEL
LIN {X 0,Y 524.017,Z 741.75,A -85,B 0,C 180,E1 -12776.551,E2 -12776.551} C_VEL
LIN {X 0,Y 523.737,Z 751.216,A -85,B 0,C 180,E1 -12776.885,E2 -12776.885} C_VEL
LIN {X 0,Y 523.398,Z 760.778,A -85,B 0,C 180,E1 -12777.315,E2 -12777.315} C_VEL
LIN {X 0,Y 523.008,Z 770.938,A -85,B 0,C 180,E1 -12777.889,E2 -12777.889} C_VEL
LIN {X 0,Y 522.549,Z 780.6,A -85,B 0,C 180,E1 -12778.56,E2 -12778.56} C_VEL
LIN {X 0,Y 522.104,Z 788.728,A -85,B 0,C 180,E1 -12779.231,E2 -12779.231} C_VEL
LIN {X 0,Y 521.553,Z 796.626,A -85,B 0,C 180,E1 -12780,E2 -12780} C_VEL
LIN {X 0,Y 520.929,Z 804.836,A -85,B 0,C 180,E1 -12780.963,E2 -12780.963} C_VEL
LIN {X 0,Y 520.542,Z 811.659,A -85,B 0,C 180,E1 -12781.928,E2 -12781.928} C_VEL
LIN {X 0,Y 520.165,Z 816.384,A -85,B 0,C 180,E1 -12782.701,E2 -12782.701} C_VEL
LIN {X 0,Y 519.93,Z 823.124,A -85,B 0,C 180,E1 -12784.11,E2 -12784.11} C_VEL
LIN {X 0,Y 519.745,Z 826.674,A -85,B 0,C 180,E1 -12785.025,E2 -12785.025} C_VEL
LIN {X 0,Y 519.588,Z 830.124,A -85,B 0,C 180,E1 -12786.191,E2 -12786.191} C_VEL
LIN {X 0,Y 519.334,Z 833.047,A -85,B 0,C 180,E1 -12787.751,E2 -12787.751} C_VEL
LIN {X 0,Y 519.335,Z 833.987,A -85,B 0,C 180,E1 -12788.532,E2 -12788.532} C_VEL
LIN {X 0,Y 519.371,Z 834.314,A -85,B 0,C 180,E1 -12790.097,E2 -12790.097} C_VEL
LIN {X 0,Y 519.321,Z 833.945,A -85,B 0,C 180,E1 -12790.884,E2 -12790.884} C_VEL
LIN {X 0,Y 519.322,Z 831.675,A -85,B 0,C 180,E1 -12792.462,E2 -12792.462} C_VEL
LIN {X 0,Y 519.428,Z 829.945,A -85,B 0,C 180,E1 -12793.252,E2 -12793.252} C_VEL
LIN {X 0,Y 519.554,Z 826.357,A -85,B 0,C 180,E1 -12794.442,E2 -12794.442} C_VEL
LIN {X 0,Y 519.701,Z 821.564,A -85,B 0,C 180,E1 -12795.638,E2 -12795.638} C_VEL
LIN {X 0,Y 519.995,Z 814.454,A -85,B 0,C 180,E1 -12796.983,E2 -12796.983} C_VEL
LIN {X 0,Y 520.244,Z 807.513,A -85,B 0,C 180,E1 -12798.039,E2 -12798.039} C_VEL
LIN {X 0,Y 520.583,Z 801.284,A -85,B 0,C 180,E1 -12798.839,E2 -12798.839} C_VEL
LIN {X 0,Y 520.937,Z 792.18,A -85,B 0,C 180,E1 -12799.809,E2 -12799.809} C_VEL
LIN {X 0,Y 521.246,Z 783.849,A -85,B 0,C 180,E1 -12800.552,E2 -12800.552} C_VEL
LIN {X 0,Y 521.717,Z 774.373,A -85,B 0,C 180,E1 -12801.253,E2 -12801.253} C_VEL
LIN {X 0,Y 522.102,Z 764.438,A -85,B 0,C 180,E1 -12801.857,E2 -12801.857} C_VEL
LIN {X 0,Y 522.444,Z 754.16,A -85,B 0,C 180,E1 -12802.358,E2 -12802.358} C_VEL
LIN {X 0,Y 522.64,Z 742.976,A -85,B 0,C 180,E1 -12802.778,E2 -12802.778} C_VEL
LIN {X 0,Y 522.894,Z 732.288,A -85,B 0,C 180,E1 -12803.067,E2 -12803.067} C_VEL
LIN {X 0,Y 523.281,Z 713.599,A -85,B 0,C 180,E1 -12803.388,E2 -12803.388} C_VEL
LIN {X 0,Y 524.181,Z 643.686,A -85,B 0,C 180,E1 -12804.51,E2 -12804.51} C_VEL
LIN {X 0,Y 521.288,Z 623.883,A -85,B 0,C 180,E1 -12804.911,E2 -12804.911} C_VEL
LIN {X 0,Y 522.039,Z 608.15,A -85,B 0,C 180,E1 -12808.009,E2 -12808.009} C_VEL
LIN {X 0,Y 522.336,Z 601.409,A -85,B 0,C 180,E1 -12809.35,E2 -12809.35} C_VEL
LIN {X 0,Y 521.348,Z 593.904,A -85,B 0,C 180,E1 -12810.901,E2 -12810.901} C_VEL
LIN {X 0,Y 521.07,Z 592.513,A -85,B 0,C 180,E1 -12811.222,E2 -12811.222} C_VEL
LIN {X 0,Y 521.002,Z 592.518,A -85,B 0,C 180,E1 -12814.378,E2 -12814.378} C_VEL
LIN {X 0,Y 521.059,Z 592.512,A -85,B 0,C 180,E1 -12816.261,E2 -12816.261} C_VEL
LIN {X 0,Y 520.981,Z 592.517,A -85,B 0,C 180,E1 -12819.19,E2 -12819.19} C_VEL
LIN {X 0,Y 521.018,Z 592.513,A -85,B 0,C 180,E1 -12821.204,E2 -12821.204} C_VEL
LIN {X 0,Y 520.998,Z 592.516,A -85,B 0,C 180,E1 -12824.557,E2 -12824.557} C_VEL
LIN {X 0,Y 521.011,Z 592.519,A -85,B 0,C 180,E1 -12827.763,E2 -12827.763} C_VEL
LIN {X 0,Y 521.032,Z 592.519,A -85,B 0,C 180,E1 -12830.02,E2 -12830.02} C_VEL
LIN {X 0,Y 521.005,Z 592.514,A -85,B 0,C 180,E1 -12832.772,E2 -12832.772} C_VEL
LIN {X 0,Y 521.028,Z 592.511,A -85,B 0,C 180,E1 -12835.089,E2 -12835.089} C_VEL
LIN {X 0,Y 521.003,Z 592.522,A -85,B 0,C 180,E1 -12837.884,E2 -12837.884} C_VEL
LIN {X 0,Y 521.015,Z 592.513,A -85,B 0,C 180,E1 -12841.054,E2 -12841.054} C_VEL
LIN {X 0,Y 521.009,Z 592.518,A -85,B 0,C 180,E1 -12843.663,E2 -12843.663} C_VEL
LIN {X 0,Y 521.009,Z 592.519,A -85,B 0,C 180,E1 -12846.214,E2 -12846.214} C_VEL
LIN {X 0,Y 521.018,Z 592.513,A -85,B 0,C 180,E1 -12848.716,E2 -12848.716} C_VEL
LIN {X 0,Y 521.008,Z 592.514,A -85,B 0,C 180,E1 -12851.176,E2 -12851.176} C_VEL
LIN {X 0,Y 521.046,Z 592.512,A -85,B 0,C 180,E1 -12853.602,E2 -12853.602} C_VEL
LIN {X 0,Y 521.107,Z 592.51,A -85,B 0,C 180,E1 -12855.998,E2 -12855.998} C_VEL
LIN {X 0,Y 521.13,Z 592.499,A -85,B 0,C 180,E1 -12859.154,E2 -12859.154} C_VEL
LIN {X 0,Y 521.16,Z 592.499,A -85,B 0,C 180,E1 -12862.276,E2 -12862.276} C_VEL
LIN {X 0,Y 521.203,Z 592.49,A -85,B 0,C 180,E1 -12864.602,E2 -12864.602} C_VEL
LIN {X 0,Y 521.177,Z 592.496,A -85,B 0,C 180,E1 -12866.348,E2 -12866.348} C_VEL
LIN {X 0,Y 521.329,Z 592.478,A -85,B 0,C 180,E1 -12869.729,E2 -12869.729} C_VEL
LIN {X 0,Y 520.676,Z 592.565,A -85,B 0,C 180,E1 -12870.373,E2 -12870.373} C_VEL
LIN {X 0,Y 517.691,Z 592.935,A -85,B 0,C 180,E1 -12871.415,E2 -12871.415} C_VEL
LIN {X 0,Y 515.166,Z 593.246,A -85,B 0,C 180,E1 -12872.255,E2 -12872.255} C_VEL
LIN {X 0,Y 514.118,Z 593.372,A -85,B 0,C 180,E1 -12872.905,E2 -12872.905} C_VEL
LIN {X 0,Y 514.055,Z 593.38,A -85,B 0,C 180,E1 -12873.125,E2 -12873.125} C_VEL
LIN {X 0,Y 514.223,Z 593.359,A -85,B 0,C 180,E1 -12874.688,E2 -12874.688} C_VEL
LIN {X 0,Y 514.108,Z 593.38,A -85,B 0,C 180,E1 -12877.83,E2 -12877.83} C_VEL
LIN {X 0,Y 514.097,Z 593.375,A -85,B 0,C 180,E1 -12881.195,E2 -12881.195} C_VEL
LIN {X 0,Y 514.076,Z 593.378,A -85,B 0,C 180,E1 -12884.673,E2 -12884.673} C_VEL
LIN {X 0,Y 513.999,Z 593.389,A -85,B 0,C 180,E1 -12887.464,E2 -12887.464} C_VEL
LIN {X 0,Y 513.992,Z 593.388,A -85,B 0,C 180,E1 -12890.751,E2 -12890.751} C_VEL
LIN {X 0,Y 513.942,Z 593.394,A -85,B 0,C 180,E1 -12893.281,E2 -12893.281} C_VEL
LIN {X 0,Y 513.942,Z 593.402,A -85,B 0,C 180,E1 -12895.908,E2 -12895.908} C_VEL
LIN {X 0,Y 513.939,Z 593.396,A -85,B 0,C 180,E1 -12898.49,E2 -12898.49} C_VEL
LIN {X 0,Y 513.973,Z 593.39,A -85,B 0,C 180,E1 -12901.189,E2 -12901.189} C_VEL
LIN {X 0,Y 513.996,Z 593.396,A -85,B 0,C 180,E1 -12903.968,E2 -12903.968} C_VEL
LIN {X 0,Y 514.003,Z 593.386,A -85,B 0,C 180,E1 -12906.841,E2 -12906.841} C_VEL
LIN {X 0,Y 513.987,Z 593.393,A -85,B 0,C 180,E1 -12910.258,E2 -12910.258} C_VEL
LIN {X 0,Y 513.947,Z 593.393,A -85,B 0,C 180,E1 -12912.956,E2 -12912.956} C_VEL
LIN {X 0,Y 513.956,Z 593.401,A -85,B 0,C 180,E1 -12915.969,E2 -12915.969} C_VEL
LIN {X 0,Y 513.966,Z 593.391,A -85,B 0,C 180,E1 -12919.145,E2 -12919.145} C_VEL
LIN {X 0,Y 514.002,Z 593.391,A -85,B 0,C 180,E1 -12922.221,E2 -12922.221} C_VEL
LIN {X 0,Y 513.982,Z 593.389,A -85,B 0,C 180,E1 -12925.085,E2 -12925.085} C_VEL
LIN {X 0,Y 513.975,Z 593.397,A -85,B 0,C 180,E1 -12927.894,E2 -12927.894} C_VEL
LIN {X 0,Y 513.973,Z 593.39,A -85,B 0,C 180,E1 -12930.714,E2 -12930.714} C_VEL
LIN {X 0,Y 513.983,Z 593.389,A -85,B 0,C 180,E1 -12933.275,E2 -12933.275} C_VEL
LIN {X 0,Y 513.967,Z 593.399,A -85,B 0,C 180,E1 -12935.936,E2 -12935.936} C_VEL
LIN {X 0,Y 513.985,Z 593.391,A -85,B 0,C 180,E1 -12938.411,E2 -12938.411} C_VEL
LIN {X 0,Y 513.963,Z 593.391,A -85,B 0,C 180,E1 -12940.909,E2 -12940.909} C_VEL
LIN {X 0,Y 513.97,Z 593.392,A -85,B 0,C 180,E1 -12943.37,E2 -12943.37} C_VEL
LIN {X 0,Y 514.063,Z 593.385,A -85,B 0,C 180,E1 -12945.803,E2 -12945.803} C_VEL
LIN {X 0,Y 514.089,Z 593.375,A -85,B 0,C 180,E1 -12949.004,E2 -12949.004} C_VEL
LIN {X 0,Y 514.114,Z 593.378,A -85,B 0,C 180,E1 -12952.17,E2 -12952.17} C_VEL
LIN {X 0,Y 514.159,Z 593.368,A -85,B 0,C 180,E1 -12954.528,E2 -12954.528} C_VEL
LIN {X 0,Y 514.05,Z 593.38,A -85,B 0,C 180,E1 -12956.876,E2 -12956.876} C_VEL
LIN {X 0,Y 514.32,Z 593.355,A -85,B 0,C 180,E1 -12960,E2 -12960} C_VEL
LIN {X 0,Y 514.214,Z 593.361,A -85,B 0,C 180,E1 -12964.688,E2 -12964.688} C_VEL
LIN {X 0,Y 514.148,Z 593.368,A -85,B 0,C 180,E1 -12967.043,E2 -12967.043} C_VEL
LIN {X 0,Y 514.086,Z 593.381,A -85,B 0,C 180,E1 -12970.203,E2 -12970.203} C_VEL
LIN {X 0,Y 514.001,Z 593.388,A -85,B 0,C 180,E1 -12972.594,E2 -12972.594} C_VEL
LIN {X 0,Y 514.033,Z 593.382,A -85,B 0,C 180,E1 -12975.005,E2 -12975.005} C_VEL
LIN {X 0,Y 513.965,Z 593.395,A -85,B 0,C 180,E1 -12978.267,E2 -12978.267} C_VEL
LIN {X 0,Y 513.941,Z 593.394,A -85,B 0,C 180,E1 -12980.754,E2 -12980.754} C_VEL
LIN {X 0,Y 513.94,Z 593.395,A -85,B 0,C 180,E1 -12983.281,E2 -12983.281} C_VEL
LIN {X 0,Y 513.942,Z 593.402,A -85,B 0,C 180,E1 -12985.907,E2 -12985.907} C_VEL
LIN {X 0,Y 513.939,Z 593.396,A -85,B 0,C 180,E1 -12988.491,E2 -12988.491} C_VEL
LIN {X 0,Y 513.911,Z 593.398,A -85,B 0,C 180,E1 -12991.193,E2 -12991.193} C_VEL
LIN {X 0,Y 513.923,Z 593.405,A -85,B 0,C 180,E1 -12993.973,E2 -12993.973} C_VEL
LIN {X 0,Y 513.942,Z 593.394,A -85,B 0,C 180,E1 -12996.846,E2 -12996.846} C_VEL
LIN {X 0,Y 513.918,Z 593.404,A -85,B 0,C 180,E1 -12999.836,E2 -12999.836} C_VEL
LIN {X 0,Y 513.945,Z 593.393,A -85,B 0,C 180,E1 -13002.956,E2 -13002.956} C_VEL
LIN {X 0,Y 513.951,Z 593.397,A -85,B 0,C 180,E1 -13006.246,E2 -13006.246} C_VEL
LIN {X 0,Y 513.918,Z 593.397,A -85,B 0,C 180,E1 -13009.14,E2 -13009.14} C_VEL
LIN {X 0,Y 513.908,Z 593.403,A -85,B 0,C 180,E1 -13012.235,E2 -13012.235} C_VEL
LIN {X 0,Y 513.913,Z 593.398,A -85,B 0,C 180,E1 -13014.863,E2 -13014.863} C_VEL
LIN {X 0,Y 513.925,Z 593.404,A -85,B 0,C 180,E1 -13017.89,E2 -13017.89} C_VEL
LIN {X 0,Y 513.969,Z 593.391,A -85,B 0,C 180,E1 -13020.715,E2 -13020.715} C_VEL
LIN {X 0,Y 513.948,Z 593.394,A -85,B 0,C 180,E1 -13023.273,E2 -13023.273} C_VEL
LIN {X 0,Y 514.023,Z 593.497,A -85,B 0,C 180,E1 -13025.472,E2 -13025.472} C_VEL
LIN {X 0,Y 516.263,Z 606.283,A -85,B 0,C 180,E1 -13027.883,E2 -13027.883} C_VEL
LIN {X 0,Y 515.636,Z 619.016,A -85,B 0,C 180,E1 -13030.147,E2 -13030.147} C_VEL
LIN {X 0,Y 514.538,Z 637.482,A -85,B 0,C 180,E1 -13033.389,E2 -13033.389} C_VEL
LIN {X 0,Y 514.118,Z 646.424,A -85,B 0,C 180,E1 -13034.947,E2 -13034.947} C_VEL
LIN {X 0,Y 517.079,Z 673.139,A -85,B 0,C 180,E1 -13035.475,E2 -13035.475} C_VEL
LIN {X 0,Y 515.959,Z 752.78,A -85,B 0,C 180,E1 -13036.782,E2 -13036.782} C_VEL
LIN {X 0,Y 515.742,Z 762.745,A -85,B 0,C 180,E1 -13037.026,E2 -13037.026} C_VEL
LIN {X 0,Y 515.399,Z 773.411,A -85,B 0,C 180,E1 -13037.391,E2 -13037.391} C_VEL
LIN {X 0,Y 515.112,Z 783.269,A -85,B 0,C 180,E1 -13037.833,E2 -13037.833} C_VEL
LIN {X 0,Y 514.773,Z 792.616,A -85,B 0,C 180,E1 -13038.352,E2 -13038.352} C_VEL
LIN {X 0,Y 514.38,Z 802.278,A -85,B 0,C 180,E1 -13039.01,E2 -13039.01} C_VEL
LIN {X 0,Y 513.889,Z 811.748,A -85,B 0,C 180,E1 -13039.794,E2 -13039.794} C_VEL
LIN {X 0,Y 513.502,Z 819.706,A -85,B 0,C 180,E1 -13040.579,E2 -13040.579} C_VEL
LIN {X 0,Y 513.105,Z 827.97,A -85,B 0,C 180,E1 -13041.562,E2 -13041.562} C_VEL
LIN {X 0,Y 512.822,Z 834.847,A -85,B 0,C 180,E1 -13042.545,E2 -13042.545} C_VEL
LIN {X 0,Y 512.656,Z 839.594,A -85,B 0,C 180,E1 -13043.331,E2 -13043.331} C_VEL
LIN {X 0,Y 512.49,Z 845.352,A -85,B 0,C 180,E1 -13044.51,E2 -13044.51} C_VEL
LIN {X 0,Y 512.378,Z 849.865,A -85,B 0,C 180,E1 -13045.688,E2 -13045.688} C_VEL
LIN {X 0,Y 512.326,Z 853.262,A -85,B 0,C 180,E1 -13046.865,E2 -13046.865} C_VEL
LIN {X 0,Y 512.326,Z 854.923,A -85,B 0,C 180,E1 -13047.649,E2 -13047.649} C_VEL
LIN {X 0,Y 512.348,Z 857.024,A -85,B 0,C 180,E1 -13049.217,E2 -13049.217} C_VEL
LIN {X 0,Y 512.325,Z 857.289,A -85,B 0,C 180,E1 -13050.784,E2 -13050.784} C_VEL
LIN {X 0,Y 512.306,Z 856.912,A -85,B 0,C 180,E1 -13051.567,E2 -13051.567} C_VEL
LIN {X 0,Y 512.334,Z 854.639,A -85,B 0,C 180,E1 -13053.135,E2 -13053.135} C_VEL
LIN {X 0,Y 512.378,Z 851.847,A -85,B 0,C 180,E1 -13054.312,E2 -13054.312} C_VEL
LIN {X 0,Y 512.523,Z 847.994,A -85,B 0,C 180,E1 -13055.49,E2 -13055.49} C_VEL
LIN {X 0,Y 512.751,Z 842.978,A -85,B 0,C 180,E1 -13056.668,E2 -13056.668} C_VEL
LIN {X 0,Y 513.008,Z 837.852,A -85,B 0,C 180,E1 -13057.65,E2 -13057.65} C_VEL
LIN {X 0,Y 513.33,Z 831.68,A -85,B 0,C 180,E1 -13058.633,E2 -13058.633} C_VEL
LIN {X 0,Y 513.85,Z 824.244,A -85,B 0,C 180,E1 -13059.613,E2 -13059.613} C_VEL
LIN {X 0,Y 514.471,Z 815.226,A -85,B 0,C 180,E1 -13060.591,E2 -13060.591} C_VEL
LIN {X 0,Y 515.033,Z 806.905,A -85,B 0,C 180,E1 -13061.348,E2 -13061.348} C_VEL
LIN {X 0,Y 515.577,Z 796.698,A -85,B 0,C 180,E1 -13062.117,E2 -13062.117} C_VEL
LIN {X 0,Y 516.075,Z 786.506,A -85,B 0,C 180,E1 -13062.742,E2 -13062.742} C_VEL
LIN {X 0,Y 516.649,Z 775.492,A -85,B 0,C 180,E1 -13063.275,E2 -13063.275} C_VEL
LIN {X 0,Y 517.121,Z 765.934,A -85,B 0,C 180,E1 -13063.637,E2 -13063.637} C_VEL
LIN {X 0,Y 517.52,Z 754.736,A -85,B 0,C 180,E1 -13063.951,E2 -13063.951} C_VEL
LIN {X 0,Y 517.997,Z 732.071,A -85,B 0,C 180,E1 -13064.362,E2 -13064.362} C_VEL
LIN {X 0,Y 519.021,Z 671.26,A -85,B 0,C 180,E1 -13065.42,E2 -13065.42} C_VEL
LIN {X 0,Y 516.692,Z 654.855,A -85,B 0,C 180,E1 -13065.819,E2 -13065.819} C_VEL
LIN {X 0,Y 514.915,Z 645.14,A -85,B 0,C 180,E1 -13066.102,E2 -13066.102} C_VEL
LIN {X 0,Y 516.282,Z 625.923,A -85,B 0,C 180,E1 -13069.62,E2 -13069.62} C_VEL
LIN {X 0,Y 517.434,Z 611.877,A -85,B 0,C 180,E1 -13072.274,E2 -13072.274} C_VEL
LIN {X 0,Y 515.833,Z 602.086,A -85,B 0,C 180,E1 -13074.337,E2 -13074.337} C_VEL
LIN {X 0,Y 513.972,Z 593.401,A -85,B 0,C 180,E1 -13076.317,E2 -13076.317} C_VEL
LIN {X 0,Y 513.968,Z 593.4,A -85,B 0,C 180,E1 -13079.381,E2 -13079.381} C_VEL
LIN {X 0,Y 513.915,Z 593.404,A -85,B 0,C 180,E1 -13082.325,E2 -13082.325} C_VEL
LIN {X 0,Y 513.938,Z 593.4,A -85,B 0,C 180,E1 -13085.141,E2 -13085.141} C_VEL
LIN {X 0,Y 513.962,Z 593.391,A -85,B 0,C 180,E1 -13087.773,E2 -13087.773} C_VEL
LIN {X 0,Y 513.921,Z 593.396,A -85,B 0,C 180,E1 -13090.86,E2 -13090.86} C_VEL
LIN {X 0,Y 513.953,Z 593.396,A -85,B 0,C 180,E1 -13093.754,E2 -13093.754} C_VEL
LIN {X 0,Y 513.957,Z 593.398,A -85,B 0,C 180,E1 -13097.045,E2 -13097.045} C_VEL
LIN {X 0,Y 513.978,Z 593.393,A -85,B 0,C 180,E1 -13100.17,E2 -13100.17} C_VEL
LIN {X 0,Y 514.01,Z 593.391,A -85,B 0,C 180,E1 -13103.514,E2 -13103.514} C_VEL
LIN {X 0,Y 513.959,Z 593.395,A -85,B 0,C 180,E1 -13106.236,E2 -13106.236} C_VEL
LIN {X 0,Y 513.963,Z 593.396,A -85,B 0,C 180,E1 -13109.158,E2 -13109.158} C_VEL
LIN {X 0,Y 513.943,Z 593.398,A -85,B 0,C 180,E1 -13111.51,E2 -13111.51} C_VEL
LIN {X 0,Y 513.949,Z 593.399,A -85,B 0,C 180,E1 -13114.143,E2 -13114.143} C_VEL
LIN {X 0,Y 513.947,Z 593.402,A -85,B 0,C 180,E1 -13116.719,E2 -13116.719} C_VEL
LIN {X 0,Y 513.999,Z 593.395,A -85,B 0,C 180,E1 -13119.249,E2 -13119.249} C_VEL
LIN {X 0,Y 513.997,Z 593.398,A -85,B 0,C 180,E1 -13122.554,E2 -13122.554} C_VEL
LIN {X 0,Y 514.067,Z 593.384,A -85,B 0,C 180,E1 -13125.803,E2 -13125.803} C_VEL
LIN {X 0,Y 514.039,Z 593.455,A -85,B 0,C 180,E1 -13126.656,E2 -13126.656} C_VEL
LIN {X 0,Y 516.009,Z 603.084,A -85,B 0,C 180,E1 -13129.045,E2 -13129.045} C_VEL
LIN {X 0,Y 516.686,Z 608.15,A -85,B 0,C 180,E1 -13130.244,E2 -13130.244} C_VEL
LIN {X 0,Y 516.277,Z 615.331,A -85,B 0,C 180,E1 -13131.81,E2 -13131.81} C_VEL
LIN {X 0,Y 515.423,Z 625.839,A -85,B 0,C 180,E1 -13134.003,E2 -13134.003} C_VEL
LIN {X 0,Y 518.724,Z 642.086,A -85,B 0,C 180,E1 -13134.455,E2 -13134.455} C_VEL
LIN {X 0,Y 519.539,Z 647.278,A -85,B 0,C 180,E1 -13134.584,E2 -13134.584} C_VEL
LIN {X 0,Y 517.88,Z 714.462,A -85,B 0,C 180,E1 -13135.734,E2 -13135.734} C_VEL
LIN {X 0,Y 517.454,Z 735.893,A -85,B 0,C 180,E1 -13136.143,E2 -13136.143} C_VEL
LIN {X 0,Y 516.981,Z 749.917,A -85,B 0,C 180,E1 -13136.602,E2 -13136.602} C_VEL
LIN {X 0,Y 516.583,Z 760.638,A -85,B 0,C 180,E1 -13137.085,E2 -13137.085} C_VEL
LIN {X 0,Y 516.159,Z 770.866,A -85,B 0,C 180,E1 -13137.667,E2 -13137.667} C_VEL
LIN {X 0,Y 515.677,Z 780.577,A -85,B 0,C 180,E1 -13138.346,E2 -13138.346} C_VEL
LIN {X 0,Y 515.136,Z 789.76,A -85,B 0,C 180,E1 -13139.123,E2 -13139.123} C_VEL
LIN {X 0,Y 514.656,Z 796.669,A -85,B 0,C 180,E1 -13139.805,E2 -13139.805} C_VEL
LIN {X 0,Y 513.966,Z 804.917,A -85,B 0,C 180,E1 -13140.781,E2 -13140.781} C_VEL
LIN {X 0,Y 513.577,Z 811.76,A -85,B 0,C 180,E1 -13141.758,E2 -13141.758} C_VEL
LIN {X 0,Y 513.09,Z 817.516,A -85,B 0,C 180,E1 -13142.738,E2 -13142.738} C_VEL
LIN {X 0,Y 512.901,Z 823.05,A -85,B 0,C 180,E1 -13143.915,E2 -13143.915} C_VEL
LIN {X 0,Y 512.667,Z 827.412,A -85,B 0,C 180,E1 -13145.095,E2 -13145.095} C_VEL
LIN {X 0,Y 512.474,Z 830.691,A -85,B 0,C 180,E1 -13146.277,E2 -13146.277} C_VEL
LIN {X 0,Y 512.351,Z 832.343,A -85,B 0,C 180,E1 -13147.067,E2 -13147.067} C_VEL
LIN {X 0,Y 512.256,Z 834.246,A -85,B 0,C 180,E1 -13148.65,E2 -13148.65} C_VEL
LIN {X 0,Y 512.274,Z 834.453,A -85,B 0,C 180,E1 -13150.109,E2 -13150.109} C_VEL
LIN {X 0,Y 512.227,Z 833.931,A -85,B 0,C 180,E1 -13151.037,E2 -13151.037} C_VEL
LIN {X 0,Y 512.204,Z 832.89,A -85,B 0,C 180,E1 -13151.837,E2 -13151.837} C_VEL
LIN {X 0,Y 512.369,Z 829.611,A -85,B 0,C 180,E1 -13153.438,E2 -13153.438} C_VEL
LIN {X 0,Y 512.505,Z 825.814,A -85,B 0,C 180,E1 -13154.645,E2 -13154.645} C_VEL
LIN {X 0,Y 512.659,Z 820.766,A -85,B 0,C 180,E1 -13155.858,E2 -13155.858} C_VEL
LIN {X 0,Y 512.893,Z 815.546,A -85,B 0,C 180,E1 -13156.871,E2 -13156.871} C_VEL
LIN {X 0,Y 513.11,Z 809.183,A -85,B 0,C 180,E1 -13157.887,E2 -13157.887} C_VEL
LIN {X 0,Y 513.516,Z 801.452,A -85,B 0,C 180,E1 -13158.902,E2 -13158.902} C_VEL
LIN {X 0,Y 513.875,Z 792.593,A -85,B 0,C 180,E1 -13159.861,E2 -13159.861} C_VEL
LIN {X 0,Y 514.21,Z 784.008,A -85,B 0,C 180,E1 -13160.638,E2 -13160.638} C_VEL
LIN {X 0,Y 514.691,Z 774.526,A -85,B 0,C 180,E1 -13161.348,E2 -13161.348} C_VEL
LIN {X 0,Y 515.085,Z 764.59,A -85,B 0,C 180,E1 -13161.96,E2 -13161.96} C_VEL
LIN {X 0,Y 515.445,Z 754.206,A -85,B 0,C 180,E1 -13162.472,E2 -13162.472} C_VEL
LIN {X 0,Y 515.626,Z 743.471,A -85,B 0,C 180,E1 -13162.884,E2 -13162.884} C_VEL
LIN {X 0,Y 515.899,Z 732.491,A -85,B 0,C 180,E1 -13163.187,E2 -13163.187} C_VEL
LIN {X 0,Y 516.309,Z 712.324,A -85,B 0,C 180,E1 -13163.538,E2 -13163.538} C_VEL
LIN {X 0,Y 517.206,Z 644.498,A -85,B 0,C 180,E1 -13164.646,E2 -13164.646} C_VEL
LIN {X 0,Y 514.254,Z 623.975,A -85,B 0,C 180,E1 -13165.083,E2 -13165.083} C_VEL
LIN {X 0,Y 515.023,Z 608.831,A -85,B 0,C 180,E1 -13168.098,E2 -13168.098} C_VEL
LIN {X 0,Y 515.282,Z 601.674,A -85,B 0,C 180,E1 -13169.543,E2 -13169.543} C_VEL
LIN {X 0,Y 514.023,Z 593.392,A -85,B 0,C 180,E1 -13171.299,E2 -13171.299} C_VEL
LIN {X 0,Y 513.955,Z 593.401,A -85,B 0,C 180,E1 -13173.97,E2 -13173.97} C_VEL
LIN {X 0,Y 513.965,Z 593.391,A -85,B 0,C 180,E1 -13176.844,E2 -13176.844} C_VEL
LIN {X 0,Y 513.989,Z 593.393,A -85,B 0,C 180,E1 -13180.257,E2 -13180.257} C_VEL
LIN {X 0,Y 513.949,Z 593.393,A -85,B 0,C 180,E1 -13182.955,E2 -13182.955} C_VEL
LIN {X 0,Y 513.958,Z 593.401,A -85,B 0,C 180,E1 -13185.968,E2 -13185.968} C_VEL
LIN {X 0,Y 513.967,Z 593.391,A -85,B 0,C 180,E1 -13189.144,E2 -13189.144} C_VEL
LIN {X 0,Y 513.961,Z 593.396,A -85,B 0,C 180,E1 -13192.226,E2 -13192.226} C_VEL
LIN {X 0,Y 513.983,Z 593.389,A -85,B 0,C 180,E1 -13195.084,E2 -13195.084} C_VEL
LIN {X 0,Y 513.974,Z 593.398,A -85,B 0,C 180,E1 -13197.893,E2 -13197.893} C_VEL
LIN {X 0,Y 513.972,Z 593.391,A -85,B 0,C 180,E1 -13200.714,E2 -13200.714} C_VEL
LIN {X 0,Y 513.982,Z 593.389,A -85,B 0,C 180,E1 -13203.274,E2 -13203.274} C_VEL
LIN {X 0,Y 513.965,Z 593.399,A -85,B 0,C 180,E1 -13205.935,E2 -13205.935} C_VEL
LIN {X 0,Y 513.982,Z 593.392,A -85,B 0,C 180,E1 -13208.411,E2 -13208.411} C_VEL
LIN {X 0,Y 513.963,Z 593.391,A -85,B 0,C 180,E1 -13210.908,E2 -13210.908} C_VEL
LIN {X 0,Y 513.99,Z 593.389,A -85,B 0,C 180,E1 -13213.37,E2 -13213.37} C_VEL
LIN {X 0,Y 514.084,Z 593.382,A -85,B 0,C 180,E1 -13215.803,E2 -13215.803} C_VEL
LIN {X 0,Y 514.084,Z 593.376,A -85,B 0,C 180,E1 -13219.003,E2 -13219.003} C_VEL
LIN {X 0,Y 514.109,Z 593.379,A -85,B 0,C 180,E1 -13222.169,E2 -13222.169} C_VEL
LIN {X 0,Y 514.223,Z 593.36,A -85,B 0,C 180,E1 -13225.312,E2 -13225.312} C_VEL
LIN {X 0,Y 514.283,Z 593.356,A -85,B 0,C 180,E1 -13229.738,E2 -13229.738} C_VEL
LIN {X 0,Y 514.103,Z 593.377,A -85,B 0,C 180,E1 -13231.561,E2 -13231.561} C_VEL
LIN {X 0,Y 514.055,Z 593.38,A -85,B 0,C 180,E1 -13233.125,E2 -13233.125} C_VEL
LIN {X 0,Y 513.458,Z 593.461,A -85,B 0,C 180,E1 -13233.78,E2 -13233.78} C_VEL
LIN {X 0,Y 510.659,Z 593.808,A -85,B 0,C 180,E1 -13234.843,E2 -13234.843} C_VEL
LIN {X 0,Y 508.247,Z 594.109,A -85,B 0,C 180,E1 -13235.699,E2 -13235.699} C_VEL
LIN {X 0,Y 507.197,Z 594.238,A -85,B 0,C 180,E1 -13236.36,E2 -13236.36} C_VEL
LIN {X 0,Y 507.105,Z 594.247,A -85,B 0,C 180,E1 -13236.584,E2 -13236.584} C_VEL
LIN {X 0,Y 506.991,Z 594.262,A -85,B 0,C 180,E1 -13239.543,E2 -13239.543} C_VEL
LIN {X 0,Y 507.008,Z 594.266,A -85,B 0,C 180,E1 -13241.96,E2 -13241.96} C_VEL
LIN {X 0,Y 506.998,Z 594.259,A -85,B 0,C 180,E1 -13245.218,E2 -13245.218} C_VEL
LIN {X 0,Y 506.94,Z 594.268,A -85,B 0,C 180,E1 -13248.529,E2 -13248.529} C_VEL
LIN {X 0,Y 506.946,Z 594.265,A -85,B 0,C 180,E1 -13251.053,E2 -13251.053} C_VEL
LIN {X 0,Y 506.909,Z 594.275,A -85,B 0,C 180,E1 -13254.22,E2 -13254.22} C_VEL
LIN {X 0,Y 506.927,Z 594.268,A -85,B 0,C 180,E1 -13257.128,E2 -13257.128} C_VEL
LIN {X 0,Y 506.923,Z 594.275,A -85,B 0,C 180,E1 -13259.83,E2 -13259.83} C_VEL
LIN {X 0,Y 506.938,Z 594.267,A -85,B 0,C 180,E1 -13262.607,E2 -13262.607} C_VEL
LIN {X 0,Y 506.941,Z 594.268,A -85,B 0,C 180,E1 -13265.473,E2 -13265.473} C_VEL
LIN {X 0,Y 506.928,Z 594.275,A -85,B 0,C 180,E1 -13268.04,E2 -13268.04} C_VEL
LIN {X 0,Y 506.94,Z 594.268,A -85,B 0,C 180,E1 -13270.542,E2 -13270.542} C_VEL
LIN {X 0,Y 506.929,Z 594.272,A -85,B 0,C 180,E1 -13273.699,E2 -13273.699} C_VEL
LIN {X 0,Y 506.929,Z 594.271,A -85,B 0,C 180,E1 -13276.302,E2 -13276.302} C_VEL
LIN {X 0,Y 506.937,Z 594.269,A -85,B 0,C 180,E1 -13279.504,E2 -13279.504} C_VEL
LIN {X 0,Y 506.956,Z 594.265,A -85,B 0,C 180,E1 -13282.56,E2 -13282.56} C_VEL
LIN {X 0,Y 506.924,Z 594.27,A -85,B 0,C 180,E1 -13285.493,E2 -13285.493} C_VEL
LIN {X 0,Y 506.923,Z 594.272,A -85,B 0,C 180,E1 -13288.328,E2 -13288.328} C_VEL
LIN {X 0,Y 506.901,Z 594.271,A -85,B 0,C 180,E1 -13291.077,E2 -13291.077} C_VEL
LIN {X 0,Y 506.903,Z 594.279,A -85,B 0,C 180,E1 -13293.919,E2 -13293.919} C_VEL
LIN {X 0,Y 506.898,Z 594.274,A -85,B 0,C 180,E1 -13296.377,E2 -13296.377} C_VEL
LIN {X 0,Y 506.948,Z 594.265,A -85,B 0,C 180,E1 -13298.947,E2 -13298.947} C_VEL
LIN {X 0,Y 506.947,Z 594.269,A -85,B 0,C 180,E1 -13302.304,E2 -13302.304} C_VEL
LIN {X 0,Y 507.021,Z 594.259,A -85,B 0,C 180,E1 -13305.602,E2 -13305.602} C_VEL
LIN {X 0,Y 507.064,Z 594.251,A -85,B 0,C 180,E1 -13308.85,E2 -13308.85} C_VEL
LIN {X 0,Y 507.077,Z 594.257,A -85,B 0,C 180,E1 -13312.06,E2 -13312.06} C_VEL
LIN {X 0,Y 507.121,Z 594.246,A -85,B 0,C 180,E1 -13314.452,E2 -13314.452} C_VEL
LIN {X 0,Y 507.03,Z 594.255,A -85,B 0,C 180,E1 -13316.833,E2 -13316.833} C_VEL
LIN {X 0,Y 507.274,Z 594.233,A -85,B 0,C 180,E1 -13320,E2 -13320} C_VEL
LIN {X 0,Y 507.143,Z 594.25,A -85,B 0,C 180,E1 -13323.96,E2 -13323.96} C_VEL
LIN {X 0,Y 507.127,Z 594.246,A -85,B 0,C 180,E1 -13326.344,E2 -13326.344} C_VEL
LIN {X 0,Y 507.041,Z 594.254,A -85,B 0,C 180,E1 -13328.741,E2 -13328.741} C_VEL
LIN {X 0,Y 507.06,Z 594.252,A -85,B 0,C 180,E1 -13331.251,E2 -13331.251} C_VEL
LIN {X 0,Y 507.017,Z 594.257,A -85,B 0,C 180,E1 -13334.749,E2 -13334.749} C_VEL
LIN {X 0,Y 506.922,Z 594.273,A -85,B 0,C 180,E1 -13337.697,E2 -13337.697} C_VEL
LIN {X 0,Y 506.911,Z 594.275,A -85,B 0,C 180,E1 -13340.209,E2 -13340.209} C_VEL
LIN {X 0,Y 506.922,Z 594.269,A -85,B 0,C 180,E1 -13342.761,E2 -13342.761} C_VEL
LIN {X 0,Y 506.875,Z 594.275,A -85,B 0,C 180,E1 -13345.365,E2 -13345.365} C_VEL
LIN {X 0,Y 506.918,Z 594.277,A -85,B 0,C 180,E1 -13348.022,E2 -13348.022} C_VEL
LIN {X 0,Y 506.892,Z 594.272,A -85,B 0,C 180,E1 -13350.749,E2 -13350.749} C_VEL
LIN {X 0,Y 506.877,Z 594.283,A -85,B 0,C 180,E1 -13353.991,E2 -13353.991} C_VEL
LIN {X 0,Y 506.92,Z 594.269,A -85,B 0,C 180,E1 -13356.734,E2 -13356.734} C_VEL
LIN {X 0,Y 506.859,Z 594.278,A -85,B 0,C 180,E1 -13359.471,E2 -13359.471} C_VEL
LIN {X 0,Y 506.922,Z 594.268,A -85,B 0,C 180,E1 -13362.918,E2 -13362.918} C_VEL
LIN {X 0,Y 506.926,Z 594.272,A -85,B 0,C 180,E1 -13366.301,E2 -13366.301} C_VEL
LIN {X 0,Y 506.88,Z 594.276,A -85,B 0,C 180,E1 -13369.498,E2 -13369.498} C_VEL
LIN {X 0,Y 506.856,Z 594.278,A -85,B 0,C 180,E1 -13372.551,E2 -13372.551} C_VEL
LIN {X 0,Y 506.881,Z 594.276,A -85,B 0,C 180,E1 -13375.489,E2 -13375.489} C_VEL
LIN {X 0,Y 506.88,Z 594.277,A -85,B 0,C 180,E1 -13378.324,E2 -13378.324} C_VEL
LIN {X 0,Y 506.894,Z 594.272,A -85,B 0,C 180,E1 -13381.077,E2 -13381.077} C_VEL
LIN {X 0,Y 506.888,Z 594.281,A -85,B 0,C 180,E1 -13383.923,E2 -13383.923} C_VEL
LIN {X 0,Y 506.975,Z 594.335,A -85,B 0,C 180,E1 -13385.35,E2 -13385.35} C_VEL
LIN {X 0,Y 509.228,Z 607.019,A -85,B 0,C 180,E1 -13387.774,E2 -13387.774} C_VEL
LIN {X 0,Y 508.825,Z 616.041,A -85,B 0,C 180,E1 -13389.403,E2 -13389.403} C_VEL
LIN {X 0,Y 507.665,Z 634.762,A -85,B 0,C 180,E1 -13392.744,E2 -13392.744} C_VEL
LIN {X 0,Y 507.103,Z 646.291,A -85,B 0,C 180,E1 -13394.785,E2 -13394.785} C_VEL
LIN {X 0,Y 510.124,Z 673.511,A -85,B 0,C 180,E1 -13395.334,E2 -13395.334} C_VEL
LIN {X 0,Y 508.938,Z 753.342,A -85,B 0,C 180,E1 -13396.672,E2 -13396.672} C_VEL
LIN {X 0,Y 508.731,Z 763.064,A -85,B 0,C 180,E1 -13396.92,E2 -13396.92} C_VEL
LIN {X 0,Y 508.413,Z 773.012,A -85,B 0,C 180,E1 -13397.266,E2 -13397.266} C_VEL
LIN {X 0,Y 508.12,Z 781.987,A -85,B 0,C 180,E1 -13397.663,E2 -13397.663} C_VEL
LIN {X 0,Y 507.678,Z 793.603,A -85,B 0,C 180,E1 -13398.325,E2 -13398.325} C_VEL
LIN {X 0,Y 507.297,Z 802.609,A -85,B 0,C 180,E1 -13398.955,E2 -13398.955} C_VEL
LIN {X 0,Y 506.809,Z 812.003,A -85,B 0,C 180,E1 -13399.75,E2 -13399.75} C_VEL
LIN {X 0,Y 506.49,Z 819.034,A -85,B 0,C 180,E1 -13400.448,E2 -13400.448} C_VEL
LIN {X 0,Y 506.035,Z 827.385,A -85,B 0,C 180,E1 -13401.443,E2 -13401.443} C_VEL
LIN {X 0,Y 505.767,Z 834.343,A -85,B 0,C 180,E1 -13402.44,E2 -13402.44} C_VEL
LIN {X 0,Y 505.555,Z 840.147,A -85,B 0,C 180,E1 -13403.437,E2 -13403.437} C_VEL
LIN {X 0,Y 505.407,Z 844.973,A -85,B 0,C 180,E1 -13404.433,E2 -13404.433} C_VEL
LIN {X 0,Y 505.286,Z 849.544,A -85,B 0,C 180,E1 -13405.628,E2 -13405.628} C_VEL
LIN {X 0,Y 505.228,Z 852.992,A -85,B 0,C 180,E1 -13406.821,E2 -13406.821} C_VEL
LIN {X 0,Y 505.231,Z 854.653,A -85,B 0,C 180,E1 -13407.616,E2 -13407.616} C_VEL
LIN {X 0,Y 505.258,Z 856.827,A -85,B 0,C 180,E1 -13409.206,E2 -13409.206} C_VEL
LIN {X 0,Y 505.236,Z 857.145,A -85,B 0,C 180,E1 -13410.795,E2 -13410.795} C_VEL
LIN {X 0,Y 505.223,Z 856.779,A -85,B 0,C 180,E1 -13411.589,E2 -13411.589} C_VEL
LIN {X 0,Y 505.234,Z 854.587,A -85,B 0,C 180,E1 -13413.179,E2 -13413.179} C_VEL
LIN {X 0,Y 505.287,Z 851.836,A -85,B 0,C 180,E1 -13414.373,E2 -13414.373} C_VEL
LIN {X 0,Y 505.456,Z 848.023,A -85,B 0,C 180,E1 -13415.567,E2 -13415.567} C_VEL
LIN {X 0,Y 505.705,Z 843.049,A -85,B 0,C 180,E1 -13416.761,E2 -13416.761} C_VEL
LIN {X 0,Y 506.045,Z 836.764,A -85,B 0,C 180,E1 -13417.956,E2 -13417.956} C_VEL
LIN {X 0,Y 506.424,Z 830.394,A -85,B 0,C 180,E1 -13418.952,E2 -13418.952} C_VEL
LIN {X 0,Y 506.996,Z 822.726,A -85,B 0,C 180,E1 -13419.945,E2 -13419.945} C_VEL
LIN {X 0,Y 507.588,Z 814.465,A -85,B 0,C 180,E1 -13420.837,E2 -13420.837} C_VEL
LIN {X 0,Y 508.151,Z 806.052,A -85,B 0,C 180,E1 -13421.603,E2 -13421.603} C_VEL
LIN {X 0,Y 508.67,Z 797.217,A -85,B 0,C 180,E1 -13422.284,E2 -13422.284} C_VEL
LIN {X 0,Y 509.209,Z 787.257,A -85,B 0,C 180,E1 -13422.916,E2 -13422.916} C_VEL
LIN {X 0,Y 509.81,Z 776.576,A -85,B 0,C 180,E1 -13423.457,E2 -13423.457} C_VEL
LIN {X 0,Y 510.341,Z 765.984,A -85,B 0,C 180,E1 -13423.873,E2 -13423.873} C_VEL
LIN {X 0,Y 510.765,Z 754.962,A -85,B 0,C 180,E1 -13424.19,E2 -13424.19} C_VEL
LIN {X 0,Y 511.179,Z 735.376,A -85,B 0,C 180,E1 -13424.558,E2 -13424.558} C_VEL
LIN {X 0,Y 512.382,Z 672.313,A -85,B 0,C 180,E1 -13425.674,E2 -13425.674} C_VEL
LIN {X 0,Y 510.228,Z 656.807,A -85,B 0,C 180,E1 -13426.062,E2 -13426.062} C_VEL
LIN {X 0,Y 507.997,Z 645.007,A -85,B 0,C 180,E1 -13426.406,E2 -13426.406} C_VEL
LIN {X 0,Y 509.28,Z 628.461,A -85,B 0,C 180,E1 -13429.483,E2 -13429.483} C_VEL
LIN {X 0,Y 510.561,Z 614.463,A -85,B 0,C 180,E1 -13432.165,E2 -13432.165} C_VEL
LIN {X 0,Y 509.814,Z 608.188,A -85,B 0,C 180,E1 -13433.481,E2 -13433.481} C_VEL
LIN {X 0,Y 508.211,Z 600.061,A -85,B 0,C 180,E1 -13435.294,E2 -13435.294} C_VEL
LIN {X 0,Y 506.941,Z 594.278,A -85,B 0,C 180,E1 -13436.683,E2 -13436.683} C_VEL
LIN {X 0,Y 506.908,Z 594.281,A -85,B 0,C 180,E1 -13439.831,E2 -13439.831} C_VEL
LIN {X 0,Y 506.892,Z 594.278,A -85,B 0,C 180,E1 -13442.61,E2 -13442.61} C_VEL
LIN {X 0,Y 506.911,Z 594.275,A -85,B 0,C 180,E1 -13445.475,E2 -13445.475} C_VEL
LIN {X 0,Y 506.888,Z 594.27,A -85,B 0,C 180,E1 -13448.033,E2 -13448.033} C_VEL
LIN {X 0,Y 506.871,Z 594.273,A -85,B 0,C 180,E1 -13450.532,E2 -13450.532} C_VEL
LIN {X 0,Y 506.929,Z 594.27,A -85,B 0,C 180,E1 -13453.699,E2 -13453.699} C_VEL
LIN {X 0,Y 506.933,Z 594.272,A -85,B 0,C 180,E1 -13457.081,E2 -13457.081} C_VEL
LIN {X 0,Y 506.942,Z 594.273,A -85,B 0,C 180,E1 -13459.504,E2 -13459.504} C_VEL
LIN {X 0,Y 506.923,Z 594.273,A -85,B 0,C 180,E1 -13462.557,E2 -13462.557} C_VEL
LIN {X 0,Y 506.93,Z 594.272,A -85,B 0,C 180,E1 -13465.493,E2 -13465.493} C_VEL
LIN {X 0,Y 506.931,Z 594.27,A -85,B 0,C 180,E1 -13468.328,E2 -13468.328} C_VEL
LIN {X 0,Y 506.905,Z 594.276,A -85,B 0,C 180,E1 -13471.077,E2 -13471.077} C_VEL
LIN {X 0,Y 506.902,Z 594.276,A -85,B 0,C 180,E1 -13473.92,E2 -13473.92} C_VEL
LIN {X 0,Y 506.901,Z 594.278,A -85,B 0,C 180,E1 -13476.376,E2 -13476.376} C_VEL
LIN {X 0,Y 506.953,Z 594.276,A -85,B 0,C 180,E1 -13478.947,E2 -13478.947} C_VEL
LIN {X 0,Y 506.951,Z 594.277,A -85,B 0,C 180,E1 -13482.304,E2 -13482.304} C_VEL
LIN {X 0,Y 507.025,Z 594.262,A -85,B 0,C 180,E1 -13485.601,E2 -13485.601} C_VEL
LIN {X 0,Y 507.005,Z 594.335,A -85,B 0,C 180,E1 -13486.315,E2 -13486.315} C_VEL
LIN {X 0,Y 509.09,Z 604.479,A -85,B 0,C 180,E1 -13488.894,E2 -13488.894} C_VEL
LIN {X 0,Y 509.796,Z 609.514,A -85,B 0,C 180,E1 -13490.11,E2 -13490.11} C_VEL
LIN {X 0,Y 509.381,Z 616.634,A -85,B 0,C 180,E1 -13491.698,E2 -13491.698} C_VEL
LIN {X 0,Y 508.552,Z 625.782,A -85,B 0,C 180,E1 -13493.674,E2 -13493.674} C_VEL
LIN {X 0,Y 511.814,Z 641.473,A -85,B 0,C 180,E1 -13494.145,E2 -13494.145} C_VEL
LIN {X 0,Y 512.87,Z 648.028,A -85,B 0,C 180,E1 -13494.317,E2 -13494.317} C_VEL
LIN {X 0,Y 511.178,Z 714.618,A -85,B 0,C 180,E1 -13495.481,E2 -13495.481} C_VEL
LIN {X 0,Y 510.736,Z 735.965,A -85,B 0,C 180,E1 -13495.895,E2 -13495.895} C_VEL
LIN {X 0,Y 510.223,Z 750.044,A -85,B 0,C 180,E1 -13496.359,E2 -13496.359} C_VEL
LIN {X 0,Y 509.784,Z 760.782,A -85,B 0,C 180,E1 -13496.849,E2 -13496.849} C_VEL
LIN {X 0,Y 509.359,Z 770.954,A -85,B 0,C 180,E1 -13497.438,E2 -13497.438} C_VEL
LIN {X 0,Y 508.83,Z 780.645,A -85,B 0,C 180,E1 -13498.126,E2 -13498.126} C_VEL
LIN {X 0,Y 508.278,Z 789.807,A -85,B 0,C 180,E1 -13498.914,E2 -13498.914} C_VEL
LIN {X 0,Y 507.576,Z 798.436,A -85,B 0,C 180,E1 -13499.802,E2 -13499.802} C_VEL
LIN {X 0,Y 507.038,Z 804.993,A -85,B 0,C 180,E1 -13500.593,E2 -13500.593} C_VEL
LIN {X 0,Y 506.597,Z 811.863,A -85,B 0,C 180,E1 -13501.584,E2 -13501.584} C_VEL
LIN {X 0,Y 506.1,Z 817.638,A -85,B 0,C 180,E1 -13502.578,E2 -13502.578} C_VEL
LIN {X 0,Y 505.861,Z 822.417,A -85,B 0,C 180,E1 -13503.572,E2 -13503.572} C_VEL
LIN {X 0,Y 505.634,Z 826.977,A -85,B 0,C 180,E1 -13504.767,E2 -13504.767} C_VEL
LIN {X 0,Y 505.48,Z 829.722,A -85,B 0,C 180,E1 -13505.728,E2 -13505.728} C_VEL
LIN {X 0,Y 505.266,Z 832.869,A -85,B 0,C 180,E1 -13507.167,E2 -13507.167} C_VEL
LIN {X 0,Y 505.152,Z 834.493,A -85,B 0,C 180,E1 -13508.773,E2 -13508.773} C_VEL
LIN {X 0,Y 505.186,Z 834.787,A -85,B 0,C 180,E1 -13509.577,E2 -13509.577} C_VEL
LIN {X 0,Y 505.139,Z 833.839,A -85,B 0,C 180,E1 -13511.194,E2 -13511.194} C_VEL
LIN {X 0,Y 505.108,Z 832.795,A -85,B 0,C 180,E1 -13512.005,E2 -13512.005} C_VEL
LIN {X 0,Y 505.3,Z 829.168,A -85,B 0,C 180,E1 -13513.63,E2 -13513.63} C_VEL
LIN {X 0,Y 505.437,Z 825.174,A -85,B 0,C 180,E1 -13514.855,E2 -13514.855} C_VEL
LIN {X 0,Y 505.522,Z 821.911,A -85,B 0,C 180,E1 -13515.675,E2 -13515.675} C_VEL
LIN {X 0,Y 505.83,Z 815.719,A -85,B 0,C 180,E1 -13516.905,E2 -13516.905} C_VEL
LIN {X 0,Y 506.049,Z 809.348,A -85,B 0,C 180,E1 -13517.937,E2 -13517.937} C_VEL
LIN {X 0,Y 506.446,Z 801.609,A -85,B 0,C 180,E1 -13518.966,E2 -13518.966} C_VEL
LIN {X 0,Y 506.826,Z 793.236,A -85,B 0,C 180,E1 -13519.892,E2 -13519.892} C_VEL
LIN {X 0,Y 507.158,Z 784.156,A -85,B 0,C 180,E1 -13520.726,E2 -13520.726} C_VEL
LIN {X 0,Y 507.662,Z 774.677,A -85,B 0,C 180,E1 -13521.446,E2 -13521.446} C_VEL
LIN {X 0,Y 508.056,Z 764.736,A -85,B 0,C 180,E1 -13522.067,E2 -13522.067} C_VEL
LIN {X 0,Y 508.414,Z 754.538,A -85,B 0,C 180,E1 -13522.579,E2 -13522.579} C_VEL
LIN {X 0,Y 508.614,Z 743.677,A -85,B 0,C 180,E1 -13523.002,E2 -13523.002} C_VEL
LIN {X 0,Y 508.892,Z 732.704,A -85,B 0,C 180,E1 -13523.31,E2 -13523.31} C_VEL
LIN {X 0,Y 509.337,Z 711.17,A -85,B 0,C 180,E1 -13523.691,E2 -13523.691} C_VEL
LIN {X 0,Y 510.203,Z 644.79,A -85,B 0,C 180,E1 -13524.795,E2 -13524.795} C_VEL
LIN {X 0,Y 507.23,Z 624.161,A -85,B 0,C 180,E1 -13525.234,E2 -13525.234} C_VEL
LIN {X 0,Y 507.99,Z 610.153,A -85,B 0,C 180,E1 -13528.058,E2 -13528.058} C_VEL
LIN {X 0,Y 508.224,Z 601.905,A -85,B 0,C 180,E1 -13529.746,E2 -13529.746} C_VEL
LIN {X 0,Y 506.988,Z 594.268,A -85,B 0,C 180,E1 -13531.391,E2 -13531.391} C_VEL
LIN {X 0,Y 506.927,Z 594.269,A -85,B 0,C 180,E1 -13534.507,E2 -13534.507} C_VEL
LIN {X 0,Y 506.922,Z 594.27,A -85,B 0,C 180,E1 -13537.443,E2 -13537.443} C_VEL
LIN {X 0,Y 506.943,Z 594.267,A -85,B 0,C 180,E1 -13540.541,E2 -13540.541} C_VEL
LIN {X 0,Y 506.931,Z 594.272,A -85,B 0,C 180,E1 -13543.698,E2 -13543.698} C_VEL
LIN {X 0,Y 506.931,Z 594.271,A -85,B 0,C 180,E1 -13546.301,E2 -13546.301} C_VEL
LIN {X 0,Y 506.938,Z 594.269,A -85,B 0,C 180,E1 -13549.503,E2 -13549.503} C_VEL
LIN {X 0,Y 506.92,Z 594.27,A -85,B 0,C 180,E1 -13552.556,E2 -13552.556} C_VEL
LIN {X 0,Y 506.924,Z 594.27,A -85,B 0,C 180,E1 -13555.492,E2 -13555.492} C_VEL
LIN {X 0,Y 506.919,Z 594.272,A -85,B 0,C 180,E1 -13558.327,E2 -13558.327} C_VEL
LIN {X 0,Y 506.9,Z 594.271,A -85,B 0,C 180,E1 -13561.077,E2 -13561.077} C_VEL
LIN {X 0,Y 506.901,Z 594.279,A -85,B 0,C 180,E1 -13563.919,E2 -13563.919} C_VEL
LIN {X 0,Y 506.896,Z 594.275,A -85,B 0,C 180,E1 -13566.376,E2 -13566.376} C_VEL
LIN {X 0,Y 506.946,Z 594.265,A -85,B 0,C 180,E1 -13568.946,E2 -13568.946} C_VEL
LIN {X 0,Y 506.965,Z 594.267,A -85,B 0,C 180,E1 -13572.304,E2 -13572.304} C_VEL
LIN {X 0,Y 507.043,Z 594.257,A -85,B 0,C 180,E1 -13575.602,E2 -13575.602} C_VEL
LIN {X 0,Y 507.06,Z 594.251,A -85,B 0,C 180,E1 -13578.849,E2 -13578.849} C_VEL
LIN {X 0,Y 507.072,Z 594.257,A -85,B 0,C 180,E1 -13582.06,E2 -13582.06} C_VEL
LIN {X 0,Y 507.194,Z 594.235,A -85,B 0,C 180,E1 -13585.247,E2 -13585.247} C_VEL
LIN {X 0,Y 507.198,Z 594.234,A -85,B 0,C 180,E1 -13589.209,E2 -13589.209} C_VEL
LIN {X 0,Y 507.198,Z 594.234,A -85,B 0,C 180,E1 -13590.791,E2 -13590.791} C_VEL
LIN {X 0,Y 507.194,Z 594.235,A -85,B 0,C 180,E1 -13594.753,E2 -13594.753} C_VEL
LIN {X 0,Y 507.105,Z 594.247,A -85,B 0,C 180,E1 -13596.584,E2 -13596.584} C_VEL
LIN {X 0,Y 506.407,Z 594.334,A -85,B 0,C 180,E1 -13597.247,E2 -13597.247} C_VEL
LIN {X 0,Y 503.489,Z 594.7,A -85,B 0,C 180,E1 -13598.323,E2 -13598.323} C_VEL
LIN {X 0,Y 501.05,Z 595.004,A -85,B 0,C 180,E1 -13599.19,E2 -13599.19} C_VEL
LIN {X 0,Y 500.029,Z 595.134,A -85,B 0,C 180,E1 -13599.86,E2 -13599.86} C_VEL
LIN {X 0,Y 499.959,Z 595.137,A -85,B 0,C 180,E1 -13600.087,E2 -13600.087} C_VEL
LIN {X 0,Y 499.965,Z 595.141,A -85,B 0,C 180,E1 -13602.131,E2 -13602.131} C_VEL
LIN {X 0,Y 500,Z 595.131,A -85,B 0,C 180,E1 -13604.849,E2 -13604.849} C_VEL
LIN {X 0,Y 499.921,Z 595.149,A -85,B 0,C 180,E1 -13607.953,E2 -13607.953} C_VEL
LIN {X 0,Y 499.901,Z 595.145,A -85,B 0,C 180,E1 -13610.505,E2 -13610.505} C_VEL
LIN {X 0,Y 499.857,Z 595.148,A -85,B 0,C 180,E1 -13613.101,E2 -13613.101} C_VEL
LIN {X 0,Y 499.898,Z 595.148,A -85,B 0,C 180,E1 -13616.267,E2 -13616.267} C_VEL
LIN {X 0,Y 499.888,Z 595.146,A -85,B 0,C 180,E1 -13619.368,E2 -13619.368} C_VEL
LIN {X 0,Y 499.903,Z 595.148,A -85,B 0,C 180,E1 -13622.17,E2 -13622.17} C_VEL
LIN {X 0,Y 499.9,Z 595.143,A -85,B 0,C 180,E1 -13625.063,E2 -13625.063} C_VEL
LIN {X 0,Y 499.881,Z 595.153,A -85,B 0,C 180,E1 -13628.064,E2 -13628.064} C_VEL
LIN {X 0,Y 499.891,Z 595.144,A -85,B 0,C 180,E1 -13630.831,E2 -13630.831} C_VEL
LIN {X 0,Y 499.878,Z 595.147,A -85,B 0,C 180,E1 -13633.362,E2 -13633.362} C_VEL
LIN {X 0,Y 499.878,Z 595.147,A -85,B 0,C 180,E1 -13636.639,E2 -13636.639} C_VEL
LIN {X 0,Y 499.883,Z 595.152,A -85,B 0,C 180,E1 -13639.868,E2 -13639.868} C_VEL
LIN {X 0,Y 499.929,Z 595.139,A -85,B 0,C 180,E1 -13642.998,E2 -13642.998} C_VEL
LIN {X 0,Y 499.869,Z 595.155,A -85,B 0,C 180,E1 -13645.91,E2 -13645.91} C_VEL
LIN {X 0,Y 499.879,Z 595.146,A -85,B 0,C 180,E1 -13648.772,E2 -13648.772} C_VEL
LIN {X 0,Y 499.899,Z 595.152,A -85,B 0,C 180,E1 -13651.974,E2 -13651.974} C_VEL
LIN {X 0,Y 499.839,Z 595.155,A -85,B 0,C 180,E1 -13654.252,E2 -13654.252} C_VEL
LIN {X 0,Y 499.86,Z 595.148,A -85,B 0,C 180,E1 -13656.899,E2 -13656.899} C_VEL
LIN {X 0,Y 499.919,Z 595.147,A -85,B 0,C 180,E1 -13659.842,E2 -13659.842} C_VEL
LIN {X 0,Y 499.908,Z 595.142,A -85,B 0,C 180,E1 -13662.888,E2 -13662.888} C_VEL
LIN {X 0,Y 499.973,Z 595.135,A -85,B 0,C 180,E1 -13665.394,E2 -13665.394} C_VEL
LIN {X 0,Y 500.039,Z 595.126,A -85,B 0,C 180,E1 -13668.691,E2 -13668.691} C_VEL
LIN {X 0,Y 500.034,Z 595.135,A -85,B 0,C 180,E1 -13671.948,E2 -13671.948} C_VEL
LIN {X 0,Y 500.085,Z 595.123,A -85,B 0,C 180,E1 -13674.374,E2 -13674.374} C_VEL
LIN {X 0,Y 500.011,Z 595.13,A -85,B 0,C 180,E1 -13676.788,E2 -13676.788} C_VEL
LIN {X 0,Y 500.228,Z 595.111,A -85,B 0,C 180,E1 -13680,E2 -13680} C_VEL
LIN {X 0,Y 500.102,Z 595.126,A -85,B 0,C 180,E1 -13684.016,E2 -13684.016} C_VEL
LIN {X 0,Y 500.082,Z 595.123,A -85,B 0,C 180,E1 -13686.434,E2 -13686.434} C_VEL
LIN {X 0,Y 499.99,Z 595.132,A -85,B 0,C 180,E1 -13688.865,E2 -13688.865} C_VEL
